LIN {X 0,Y 173.444,Z 1036.446,A -85,B 0,C 180,E1 -27586.228,E2 -27586.228} C_VEL
LIN {X 0,Y 162.464,Z 1044.017,A -85,B 0,C 180,E1 -27593.346,E2 -27593.346} C_VEL
LIN {X 0,Y 153.982,Z 1050.121,A -85,B 0,C 180,E1 -27601.28,E2 -27601.28} C_VEL
LIN {X 0,Y 148.005,Z 1054.743,A -85,B 0,C 180,E1 -27610.258,E2 -27610.258} C_VEL
LIN {X 0,Y 145.243,Z 1057.412,A -85,B 0,C 180,E1 -27618.081,E2 -27618.081} C_VEL
LIN {X 0,Y 144.199,Z 1058.976,A -85,B 0,C 180,E1 -27625.626,E2 -27625.626} C_VEL
LIN {X 0,Y 144.037,Z 1059.569,A -85,B 0,C 180,E1 -27632.387,E2 -27632.387} C_VEL
LIN {X 0,Y 144.314,Z 1059.398,A -85,B 0,C 180,E1 -27639.572,E2 -27639.572} C_VEL
LIN {X 0,Y 146.072,Z 1057.914,A -85,B 0,C 180,E1 -27648.767,E2 -27648.767} C_VEL
LIN {X 0,Y 149.888,Z 1055.271,A -85,B 0,C 180,E1 -27656.976,E2 -27656.976} C_VEL
LIN {X 0,Y 156.774,Z 1051.046,A -85,B 0,C 180,E1 -27665.478,E2 -27665.478} C_VEL
LIN {X 0,Y 166.876,Z 1044.865,A -85,B 0,C 180,E1 -27673.556,E2 -27673.556} C_VEL
LIN {X 0,Y 177.931,Z 1038.053,A -85,B 0,C 180,E1 -27679.841,E2 -27679.841} C_VEL
LIN {X 0,Y 192.704,Z 1028.454,A -85,B 0,C 180,E1 -27686.119,E2 -27686.119} C_VEL
LIN {X 0,Y 206.466,Z 1018.863,A -85,B 0,C 180,E1 -27690.659,E2 -27690.659} C_VEL
LIN {X 0,Y 223.283,Z 1006.192,A -85,B 0,C 180,E1 -27695.106,E2 -27695.106} C_VEL
LIN {X 0,Y 238.041,Z 993.951,A -85,B 0,C 180,E1 -27698.306,E2 -27698.306} C_VEL
LIN {X 0,Y 254.411,Z 979.174,A -85,B 0,C 180,E1 -27701.295,E2 -27701.295} C_VEL
LIN {X 0,Y 269.808,Z 963.547,A -85,B 0,C 180,E1 -27703.706,E2 -27703.706} C_VEL
LIN {X 0,Y 285.132,Z 946.472,A -85,B 0,C 180,E1 -27705.79,E2 -27705.79} C_VEL
LIN {X 0,Y 299.537,Z 928.245,A -85,B 0,C 180,E1 -27707.528,E2 -27707.528} C_VEL
LIN {X 0,Y 312.45,Z 910.056,A -85,B 0,C 180,E1 -27708.93,E2 -27708.93} C_VEL
LIN {X 0,Y 325.685,Z 888.747,A -85,B 0,C 180,E1 -27710.233,E2 -27710.233} C_VEL
LIN {X 0,Y 335.946,Z 869.895,A -85,B 0,C 180,E1 -27711.169,E2 -27711.169} C_VEL
LIN {X 0,Y 346.944,Z 846.425,A -85,B 0,C 180,E1 -27712.112,E2 -27712.112} C_VEL
LIN {X 0,Y 354.795,Z 826.568,A -85,B 0,C 180,E1 -27712.753,E2 -27712.753} C_VEL
LIN {X 0,Y 362.673,Z 802.827,A -85,B 0,C 180,E1 -27713.362,E2 -27713.362} C_VEL
LIN {X 0,Y 368.63,Z 779.656,A -85,B 0,C 180,E1 -27713.815,E2 -27713.815} C_VEL
LIN {X 0,Y 373.408,Z 755.336,A -85,B 0,C 180,E1 -27714.19,E2 -27714.19} C_VEL
LIN {X 0,Y 379.555,Z 704.729,A -85,B 0,C 180,E1 -27714.844,E2 -27714.844} C_VEL
LIN {X 0,Y 386.488,Z 644.435,A -85,B 0,C 180,E1 -27715.615,E2 -27715.615} C_VEL
LIN {X 0,Y 385.979,Z 642.999,A -85,B 0,C 180,E1 -27716.881,E2 -27716.881} C_VEL
LIN {X 0,Y 385.387,Z 640.321,A -85,B 0,C 180,E1 -27720.892,E2 -27720.892} C_VEL
LIN {X 0,Y 386.259,Z 643.666,A -85,B 0,C 180,E1 -27725.496,E2 -27725.496} C_VEL
LIN {X 0,Y 386.489,Z 644.784,A -85,B 0,C 180,E1 -27726.121,E2 -27726.121} C_VEL
LIN {X 0,Y 373.686,Z 754.037,A -85,B 0,C 180,E1 -27727.517,E2 -27727.517} C_VEL
LIN {X 0,Y 368.823,Z 780.194,A -85,B 0,C 180,E1 -27727.896,E2 -27727.896} C_VEL
LIN {X 0,Y 363.895,Z 799.826,A -85,B 0,C 180,E1 -27728.218,E2 -27728.218} C_VEL
LIN {X 0,Y 361.672,Z 807.261,A -85,B 0,C 180,E1 -27728.183,E2 -27728.183} C_VEL
LIN {X 0,Y 354.681,Z 825.951,A -85,B 0,C 180,E1 -27727.636,E2 -27727.636} C_VEL
LIN {X 0,Y 351.901,Z 833.043,A -85,B 0,C 180,E1 -27727.655,E2 -27727.655} C_VEL
LIN {X 0,Y 341.59,Z 857.457,A -85,B 0,C 180,E1 -27728.357,E2 -27728.357} C_VEL
LIN {X 0,Y 331.506,Z 877.698,A -85,B 0,C 180,E1 -27729.106,E2 -27729.106} C_VEL
LIN {X 0,Y 318.47,Z 900.334,A -85,B 0,C 180,E1 -27730.171,E2 -27730.171} C_VEL
LIN {X 0,Y 306.359,Z 918.658,A -85,B 0,C 180,E1 -27731.256,E2 -27731.256} C_VEL
LIN {X 0,Y 292.091,Z 937.956,A -85,B 0,C 180,E1 -27732.679,E2 -27732.679} C_VEL
LIN {X 0,Y 277.137,Z 955.733,A -85,B 0,C 180,E1 -27734.366,E2 -27734.366} C_VEL
LIN {X 0,Y 260.71,Z 973.388,A -85,B 0,C 180,E1 -27736.501,E2 -27736.501} C_VEL
LIN {X 0,Y 244.275,Z 989.022,A -85,B 0,C 180,E1 -27738.994,E2 -27738.994} C_VEL
LIN {X 0,Y 227.573,Z 1003.58,A -85,B 0,C 180,E1 -27742.017,E2 -27742.017} C_VEL
LIN {X 0,Y 210.824,Z 1016.635,A -85,B 0,C 180,E1 -27745.694,E2 -27745.694} C_VEL
LIN {X 0,Y 195.09,Z 1028.025,A -85,B 0,C 180,E1 -27749.983,E2 -27749.983} C_VEL
LIN {X 0,Y 179.302,Z 1038.497,A -85,B 0,C 180,E1 -27755.494,E2 -27755.494} C_VEL
LIN {X 0,Y 166.53,Z 1046.54,A -85,B 0,C 180,E1 -27761.363,E2 -27761.363} C_VEL
LIN {X 0,Y 153.385,Z 1054.528,A -85,B 0,C 180,E1 -27769.807,E2 -27769.807} C_VEL
LIN {X 0,Y 145.319,Z 1059.505,A -85,B 0,C 180,E1 -27777.541,E2 -27777.541} C_VEL
LIN {X 0,Y 139.028,Z 1063.816,A -85,B 0,C 180,E1 -27787.593,E2 -27787.593} C_VEL
LIN {X 0,Y 136.508,Z 1066.001,A -85,B 0,C 180,E1 -27796.444,E2 -27796.444} C_VEL
LIN {X 0,Y 135.999,Z 1066.928,A -85,B 0,C 180,E1 -27804.092,E2 -27804.092} C_VEL
LIN {X 0,Y 136.059,Z 1067.021,A -85,B 0,C 180,E1 -27810,E2 -27810} C_VEL
LIN {X 0,Y 136.006,Z 1066.417,A -85,B 0,C 180,E1 -27816.755,E2 -27816.755} C_VEL
LIN {X 0,Y 136.711,Z 1064.717,A -85,B 0,C 180,E1 -27824.832,E2 -27824.832} C_VEL
LIN {X 0,Y 139.354,Z 1061.814,A -85,B 0,C 180,E1 -27833.302,E2 -27833.302} C_VEL
LIN {X 0,Y 145.833,Z 1056.613,A -85,B 0,C 180,E1 -27843.265,E2 -27843.265} C_VEL
LIN {X 0,Y 154.501,Z 1050.4,A -85,B 0,C 180,E1 -27851.309,E2 -27851.309} C_VEL
LIN {X 0,Y 166.227,Z 1042.388,A -85,B 0,C 180,E1 -27858.755,E2 -27858.755} C_VEL
LIN {X 0,Y 179.96,Z 1032.608,A -85,B 0,C 180,E1 -27865.09,E2 -27865.09} C_VEL
LIN {X 0,Y 195.382,Z 1021.235,A -85,B 0,C 180,E1 -27870.458,E2 -27870.458} C_VEL
LIN {X 0,Y 211.129,Z 1008.531,A -85,B 0,C 180,E1 -27874.771,E2 -27874.771} C_VEL
LIN {X 0,Y 227.067,Z 994.761,A -85,B 0,C 180,E1 -27878.301,E2 -27878.301} C_VEL
LIN {X 0,Y 243.473,Z 978.966,A -85,B 0,C 180,E1 -27881.317,E2 -27881.317} C_VEL
LIN {X 0,Y 258.429,Z 963.247,A -85,B 0,C 180,E1 -27883.645,E2 -27883.645} C_VEL
LIN {X 0,Y 273.92,Z 944.994,A -85,B 0,C 180,E1 -27885.732,E2 -27885.732} C_VEL
LIN {X 0,Y 287.009,Z 927.872,A -85,B 0,C 180,E1 -27887.283,E2 -27887.283} C_VEL
LIN {X 0,Y 301.23,Z 906.903,A -85,B 0,C 180,E1 -27888.775,E2 -27888.775} C_VEL
LIN {X 0,Y 312.372,Z 888.252,A -85,B 0,C 180,E1 -27889.832,E2 -27889.832} C_VEL
LIN {X 0,Y 324.093,Z 865.864,A -85,B 0,C 180,E1 -27890.845,E2 -27890.845} C_VEL
LIN {X 0,Y 333.067,Z 845.762,A -85,B 0,C 180,E1 -27891.564,E2 -27891.564} C_VEL
LIN {X 0,Y 341.865,Z 822.855,A -85,B 0,C 180,E1 -27892.213,E2 -27892.213} C_VEL
LIN {X 0,Y 349.212,Z 798.837,A -85,B 0,C 180,E1 -27892.723,E2 -27892.723} C_VEL
LIN {X 0,Y 355.105,Z 774.615,A -85,B 0,C 180,E1 -27893.129,E2 -27893.129} C_VEL
LIN {X 0,Y 359.226,Z 749.857,A -85,B 0,C 180,E1 -27893.486,E2 -27893.486} C_VEL
LIN {X 0,Y 371.93,Z 639.67,A -85,B 0,C 180,E1 -27894.91,E2 -27894.91} C_VEL
LIN {X 0,Y 370.985,Z 636.993,A -85,B 0,C 180,E1 -27897.065,E2 -27897.065} C_VEL
LIN {X 0,Y 370.365,Z 634.188,A -85,B 0,C 180,E1 -27901.392,E2 -27901.392} C_VEL
LIN {X 0,Y 371.309,Z 637.843,A -85,B 0,C 180,E1 -27906.184,E2 -27906.184} C_VEL
LIN {X 0,Y 371.884,Z 639.748,A -85,B 0,C 180,E1 -27907.457,E2 -27907.457} C_VEL
LIN {X 0,Y 358.891,Z 751.554,A -85,B 0,C 180,E1 -27908.9,E2 -27908.9} C_VEL
LIN {X 0,Y 354.116,Z 777.471,A -85,B 0,C 180,E1 -27909.3,E2 -27909.3} C_VEL
LIN {X 0,Y 348.715,Z 799.063,A -85,B 0,C 180,E1 -27909.723,E2 -27909.723} C_VEL
LIN {X 0,Y 340.54,Z 824.701,A -85,B 0,C 180,E1 -27910.384,E2 -27910.384} C_VEL
LIN {X 0,Y 332.636,Z 845.015,A -85,B 0,C 180,E1 -27911.055,E2 -27911.055} C_VEL
LIN {X 0,Y 322.011,Z 868.172,A -85,B 0,C 180,E1 -27912.008,E2 -27912.008} C_VEL
LIN {X 0,Y 311.508,Z 887.711,A -85,B 0,C 180,E1 -27913.007,E2 -27913.007} C_VEL
LIN {X 0,Y 299.205,Z 907.957,A -85,B 0,C 180,E1 -27914.274,E2 -27914.274} C_VEL
LIN {X 0,Y 285.765,Z 927.152,A -85,B 0,C 180,E1 -27915.799,E2 -27915.799} C_VEL
LIN {X 0,Y 271.231,Z 945.815,A -85,B 0,C 180,E1 -27917.645,E2 -27917.645} C_VEL
LIN {X 0,Y 256.135,Z 962.851,A -85,B 0,C 180,E1 -27919.813,E2 -27919.813} C_VEL
LIN {X 0,Y 241.033,Z 978.385,A -85,B 0,C 180,E1 -27922.319,E2 -27922.319} C_VEL
LIN {X 0,Y 224.836,Z 993.303,A -85,B 0,C 180,E1 -27925.474,E2 -27925.474} C_VEL
LIN {X 0,Y 210.146,Z 1005.718,A -85,B 0,C 180,E1 -27928.898,E2 -27928.898} C_VEL
LIN {X 0,Y 193.459,Z 1018.601,A -85,B 0,C 180,E1 -27933.682,E2 -27933.682} C_VEL
LIN {X 0,Y 180.153,Z 1028.144,A -85,B 0,C 180,E1 -27938.502,E2 -27938.502} C_VEL
LIN {X 0,Y 165.451,Z 1038.099,A -85,B 0,C 180,E1 -27945.49,E2 -27945.49} C_VEL
LIN {X 0,Y 155.106,Z 1044.871,A -85,B 0,C 180,E1 -27952.236,E2 -27952.236} C_VEL
LIN {X 0,Y 145.923,Z 1051.053,A -85,B 0,C 180,E1 -27960.889,E2 -27960.889} C_VEL
LIN {X 0,Y 140.019,Z 1055.292,A -85,B 0,C 180,E1 -27969.954,E2 -27969.954} C_VEL
LIN {X 0,Y 137.097,Z 1057.973,A -85,B 0,C 180,E1 -27978.643,E2 -27978.643} C_VEL
LIN {X 0,Y 136.125,Z 1059.517,A -85,B 0,C 180,E1 -27987.474,E2 -27987.474} C_VEL
LIN {X 0,Y 136.078,Z 1059.854,A -85,B 0,C 180,E1 -27995.059,E2 -27995.059} C_VEL
LIN {X 0,Y 136.713,Z 1059.293,A -85,B 0,C 180,E1 -28003.105,E2 -28003.105} C_VEL
LIN {X 0,Y 138.991,Z 1057.679,A -85,B 0,C 180,E1 -28011.524,E2 -28011.524} C_VEL
LIN {X 0,Y 143.709,Z 1054.848,A -85,B 0,C 180,E1 -28020.063,E2 -28020.063} C_VEL
LIN {X 0,Y 152.977,Z 1049.573,A -85,B 0,C 180,E1 -28029.833,E2 -28029.833} C_VEL
LIN {X 0,Y 163.062,Z 1043.85,A -85,B 0,C 180,E1 -28036.862,E2 -28036.862} C_VEL
LIN {X 0,Y 177.76,Z 1035.167,A -85,B 0,C 180,E1 -28044.197,E2 -28044.197} C_VEL
LIN {X 0,Y 191.676,Z 1026.338,A -85,B 0,C 180,E1 -28049.399,E2 -28049.399} C_VEL
LIN {X 0,Y 208.569,Z 1014.772,A -85,B 0,C 180,E1 -28054.327,E2 -28054.327} C_VEL
LIN {X 0,Y 224.273,Z 1002.903,A -85,B 0,C 180,E1 -28058.006,E2 -28058.006} C_VEL
LIN {X 0,Y 240.811,Z 989.282,A -85,B 0,C 180,E1 -28061.208,E2 -28061.208} C_VEL
LIN {X 0,Y 256.218,Z 975.058,A -85,B 0,C 180,E1 -28063.743,E2 -28063.743} C_VEL
LIN {X 0,Y 271.177,Z 959.936,A -85,B 0,C 180,E1 -28065.869,E2 -28065.869} C_VEL
LIN {X 0,Y 286.867,Z 942.134,A -85,B 0,C 180,E1 -28067.826,E2 -28067.826} C_VEL
LIN {X 0,Y 299.674,Z 925.914,A -85,B 0,C 180,E1 -28069.253,E2 -28069.253} C_VEL
LIN {X 0,Y 314.092,Z 905.408,A -85,B 0,C 180,E1 -28070.702,E2 -28070.702} C_VEL
LIN {X 0,Y 325.346,Z 887.102,A -85,B 0,C 180,E1 -28071.732,E2 -28071.732} C_VEL
LIN {X 0,Y 336.695,Z 866.245,A -85,B 0,C 180,E1 -28072.697,E2 -28072.697} C_VEL
LIN {X 0,Y 346.692,Z 844.499,A -85,B 0,C 180,E1 -28073.498,E2 -28073.498} C_VEL
LIN {X 0,Y 354.828,Z 823.837,A -85,B 0,C 180,E1 -28074.12,E2 -28074.12} C_VEL
LIN {X 0,Y 362.88,Z 798.729,A -85,B 0,C 180,E1 -28074.711,E2 -28074.711} C_VEL
LIN {X 0,Y 368.398,Z 776.886,A -85,B 0,C 180,E1 -28075.103,E2 -28075.103} C_VEL
LIN {X 0,Y 373.276,Z 750.254,A -85,B 0,C 180,E1 -28075.481,E2 -28075.481} C_VEL
LIN {X 0,Y 385.06,Z 651.072,A -85,B 0,C 180,E1 -28076.725,E2 -28076.725} C_VEL
LIN {X 0,Y 384.406,Z 648.313,A -85,B 0,C 180,E1 -28080.894,E2 -28080.894} C_VEL
LIN {X 0,Y 385.072,Z 651.262,A -85,B 0,C 180,E1 -28085.014,E2 -28085.014} C_VEL
LIN {X 0,Y 372.858,Z 753.848,A -85,B 0,C 180,E1 -28086.29,E2 -28086.29} C_VEL
LIN {X 0,Y 367.945,Z 779.986,A -85,B 0,C 180,E1 -28086.654,E2 -28086.654} C_VEL
LIN {X 0,Y 362.317,Z 801.977,A -85,B 0,C 180,E1 -28087,E2 -28087} C_VEL
LIN {X 0,Y 354.003,Z 827.41,A -85,B 0,C 180,E1 -28087.516,E2 -28087.516} C_VEL
LIN {X 0,Y 351.901,Z 833.043,A -85,B 0,C 180,E1 -28087.655,E2 -28087.655} C_VEL
LIN {X 0,Y 348.96,Z 840.283,A -85,B 0,C 180,E1 -28087.682,E2 -28087.682} C_VEL
LIN {X 0,Y 340.298,Z 858.245,A -85,B 0,C 180,E1 -28087.209,E2 -28087.209} C_VEL
LIN {X 0,Y 336.89,Z 865.113,A -85,B 0,C 180,E1 -28087.266,E2 -28087.266} C_VEL
LIN {X 0,Y 325.209,Z 886.908,A -85,B 0,C 180,E1 -28088.1,E2 -28088.1} C_VEL
LIN {X 0,Y 313.827,Z 905.472,A -85,B 0,C 180,E1 -28088.997,E2 -28088.997} C_VEL
LIN {X 0,Y 299.256,Z 926.414,A -85,B 0,C 180,E1 -28090.264,E2 -28090.264} C_VEL
LIN {X 0,Y 285.785,Z 943.458,A -85,B 0,C 180,E1 -28091.579,E2 -28091.579} C_VEL
LIN {X 0,Y 270.221,Z 961.244,A -85,B 0,C 180,E1 -28093.303,E2 -28093.303} C_VEL
LIN {X 0,Y 254.044,Z 977.534,A -85,B 0,C 180,E1 -28095.357,E2 -28095.357} C_VEL
LIN {X 0,Y 238.257,Z 992.011,A -85,B 0,C 180,E1 -28097.703,E2 -28097.703} C_VEL
LIN {X 0,Y 220.432,Z 1006.67,A -85,B 0,C 180,E1 -28100.864,E2 -28100.864} C_VEL
LIN {X 0,Y 204.985,Z 1018.231,A -85,B 0,C 180,E1 -28104.194,E2 -28104.194} C_VEL
LIN {X 0,Y 186.511,Z 1030.839,A -85,B 0,C 180,E1 -28109.2,E2 -28109.2} C_VEL
LIN {X 0,Y 171.931,Z 1039.978,A -85,B 0,C 180,E1 -28114.328,E2 -28114.328} C_VEL
LIN {X 0,Y 156.524,Z 1049.055,A -85,B 0,C 180,E1 -28121.634,E2 -28121.634} C_VEL
LIN {X 0,Y 145.248,Z 1055.417,A -85,B 0,C 180,E1 -28129.222,E2 -28129.222} C_VEL
LIN {X 0,Y 135.786,Z 1060.915,A -85,B 0,C 180,E1 -28138.972,E2 -28138.972} C_VEL
LIN {X 0,Y 130.572,Z 1064.21,A -85,B 0,C 180,E1 -28148.434,E2 -28148.434} C_VEL
LIN {X 0,Y 128.359,Z 1066.085,A -85,B 0,C 180,E1 -28157.402,E2 -28157.402} C_VEL
LIN {X 0,Y 128.002,Z 1066.818,A -85,B 0,C 180,E1 -28165.52,E2 -28165.52} C_VEL
LIN {X 0,Y 128.037,Z 1066.713,A -85,B 0,C 180,E1 -28171.79,E2 -28171.79} C_VEL
LIN {X 0,Y 128.044,Z 1065.979,A -85,B 0,C 180,E1 -28178.532,E2 -28178.532} C_VEL
LIN {X 0,Y 129.155,Z 1064.128,A -85,B 0,C 180,E1 -28187.109,E2 -28187.109} C_VEL
LIN {X 0,Y 133.454,Z 1060.36,A -85,B 0,C 180,E1 -28197.68,E2 -28197.68} C_VEL
LIN {X 0,Y 140.894,Z 1055.047,A -85,B 0,C 180,E1 -28207.101,E2 -28207.101} C_VEL
LIN {X 0,Y 151.918,Z 1047.938,A -85,B 0,C 180,E1 -28215.841,E2 -28215.841} C_VEL
LIN {X 0,Y 165.139,Z 1039.209,A -85,B 0,C 180,E1 -28223.057,E2 -28223.057} C_VEL
LIN {X 0,Y 179.785,Z 1029.321,A -85,B 0,C 180,E1 -28228.924,E2 -28228.924} C_VEL
LIN {X 0,Y 195.964,Z 1017.429,A -85,B 0,C 180,E1 -28233.899,E2 -28233.899} C_VEL
LIN {X 0,Y 211.756,Z 1004.997,A -85,B 0,C 180,E1 -28237.743,E2 -28237.743} C_VEL
LIN {X 0,Y 228.856,Z 990.097,A -85,B 0,C 180,E1 -28241.137,E2 -28241.137} C_VEL
LIN {X 0,Y 243.866,Z 975.771,A -85,B 0,C 180,E1 -28243.625,E2 -28243.625} C_VEL
LIN {X 0,Y 260.896,Z 957.673,A -85,B 0,C 180,E1 -28246.028,E2 -28246.028} C_VEL
LIN {X 0,Y 274.295,Z 941.809,A -85,B 0,C 180,E1 -28247.672,E2 -28247.672} C_VEL
LIN {X 0,Y 289.489,Z 921.719,A -85,B 0,C 180,E1 -28249.313,E2 -28249.313} C_VEL
LIN {X 0,Y 302.091,Z 902.766,A -85,B 0,C 180,E1 -28250.522,E2 -28250.522} C_VEL
LIN {X 0,Y 314.82,Z 881.085,A -85,B 0,C 180,E1 -28251.628,E2 -28251.628} C_VEL
LIN {X 0,Y 325.282,Z 860.292,A -85,B 0,C 180,E1 -28252.454,E2 -28252.454} C_VEL
LIN {X 0,Y 334.797,Z 838.537,A -85,B 0,C 180,E1 -28253.139,E2 -28253.139} C_VEL
LIN {X 0,Y 343.033,Z 815.564,A -85,B 0,C 180,E1 -28253.701,E2 -28253.701} C_VEL
LIN {X 0,Y 349.627,Z 793.272,A -85,B 0,C 180,E1 -28254.123,E2 -28254.123} C_VEL
LIN {X 0,Y 355.299,Z 767.873,A -85,B 0,C 180,E1 -28254.509,E2 -28254.509} C_VEL
LIN {X 0,Y 358.865,Z 745.266,A -85,B 0,C 180,E1 -28254.818,E2 -28254.818} C_VEL
LIN {X 0,Y 370.36,Z 646.203,A -85,B 0,C 180,E1 -28256.091,E2 -28256.091} C_VEL
LIN {X 0,Y 369.892,Z 644.775,A -85,B 0,C 180,E1 -28257.366,E2 -28257.366} C_VEL
LIN {X 0,Y 369.384,Z 642.181,A -85,B 0,C 180,E1 -28261.396,E2 -28261.396} C_VEL
LIN {X 0,Y 370.228,Z 645.651,A -85,B 0,C 180,E1 -28265.968,E2 -28265.968} C_VEL
LIN {X 0,Y 370.338,Z 646.293,A -85,B 0,C 180,E1 -28266.307,E2 -28266.307} C_VEL
LIN {X 0,Y 357.88,Z 751.789,A -85,B 0,C 180,E1 -28267.631,E2 -28267.631} C_VEL
LIN {X 0,Y 353.035,Z 777.762,A -85,B 0,C 180,E1 -28268.015,E2 -28268.015} C_VEL
LIN {X 0,Y 347.557,Z 799.413,A -85,B 0,C 180,E1 -28268.42,E2 -28268.42} C_VEL
LIN {X 0,Y 339.664,Z 824.008,A -85,B 0,C 180,E1 -28269.021,E2 -28269.021} C_VEL
LIN {X 0,Y 331.666,Z 844.431,A -85,B 0,C 180,E1 -28269.66,E2 -28269.66} C_VEL
LIN {X 0,Y 321.374,Z 866.861,A -85,B 0,C 180,E1 -28270.527,E2 -28270.527} C_VEL
LIN {X 0,Y 310.217,Z 887.437,A -85,B 0,C 180,E1 -28271.521,E2 -28271.521} C_VEL
LIN {X 0,Y 297.782,Z 907.691,A -85,B 0,C 180,E1 -28272.725,E2 -28272.725} C_VEL
LIN {X 0,Y 284.128,Z 926.943,A -85,B 0,C 180,E1 -28274.181,E2 -28274.181} C_VEL
LIN {X 0,Y 269.735,Z 945.158,A -85,B 0,C 180,E1 -28275.896,E2 -28275.896} C_VEL
LIN {X 0,Y 254.375,Z 962.289,A -85,B 0,C 180,E1 -28277.965,E2 -28277.965} C_VEL
LIN {X 0,Y 239.451,Z 977.364,A -85,B 0,C 180,E1 -28280.279,E2 -28280.279} C_VEL
LIN {X 0,Y 222.273,Z 992.933,A -85,B 0,C 180,E1 -28283.41,E2 -28283.41} C_VEL
LIN {X 0,Y 207.108,Z 1005.405,A -85,B 0,C 180,E1 -28286.728,E2 -28286.728} C_VEL
LIN {X 0,Y 189.492,Z 1018.593,A -85,B 0,C 180,E1 -28291.493,E2 -28291.493} C_VEL
LIN {X 0,Y 175.853,Z 1027.98,A -85,B 0,C 180,E1 -28296.157,E2 -28296.157} C_VEL
LIN {X 0,Y 160.888,Z 1037.679,A -85,B 0,C 180,E1 -28302.832,E2 -28302.832} C_VEL
LIN {X 0,Y 149.223,Z 1044.838,A -85,B 0,C 180,E1 -28309.965,E2 -28309.965} C_VEL
LIN {X 0,Y 139.232,Z 1051.1,A -85,B 0,C 180,E1 -28318.864,E2 -28318.864} C_VEL
LIN {X 0,Y 132.661,Z 1055.377,A -85,B 0,C 180,E1 -28328.326,E2 -28328.326} C_VEL
LIN {X 0,Y 129.421,Z 1057.985,A -85,B 0,C 180,E1 -28337.053,E2 -28337.053} C_VEL
LIN {X 0,Y 128.164,Z 1059.622,A -85,B 0,C 180,E1 -28346.422,E2 -28346.422} C_VEL
LIN {X 0,Y 128.058,Z 1060.074,A -85,B 0,C 180,E1 -28354.03,E2 -28354.03} C_VEL
LIN {X 0,Y 128.626,Z 1059.693,A -85,B 0,C 180,E1 -28362.572,E2 -28362.572} C_VEL
LIN {X 0,Y 131.235,Z 1057.989,A -85,B 0,C 180,E1 -28372.393,E2 -28372.393} C_VEL
LIN {X 0,Y 136.337,Z 1055.198,A -85,B 0,C 180,E1 -28381.38,E2 -28381.38} C_VEL
LIN {X 0,Y 146.26,Z 1050.004,A -85,B 0,C 180,E1 -28391.539,E2 -28391.539} C_VEL
LIN {X 0,Y 157.505,Z 1044.026,A -85,B 0,C 180,E1 -28399.065,E2 -28399.065} C_VEL
LIN {X 0,Y 172.914,Z 1035.402,A -85,B 0,C 180,E1 -28406.376,E2 -28406.376} C_VEL
LIN {X 0,Y 187.59,Z 1026.49,A -85,B 0,C 180,E1 -28411.58,E2 -28411.58} C_VEL
LIN {X 0,Y 205.337,Z 1014.749,A -85,B 0,C 180,E1 -28416.465,E2 -28416.465} C_VEL
LIN {X 0,Y 221.332,Z 1003.013,A -85,B 0,C 180,E1 -28419.995,E2 -28419.995} C_VEL
LIN {X 0,Y 239.151,Z 988.614,A -85,B 0,C 180,E1 -28423.232,E2 -28423.232} C_VEL
LIN {X 0,Y 254.925,Z 974.31,A -85,B 0,C 180,E1 -28425.651,E2 -28425.651} C_VEL
LIN {X 0,Y 271.109,Z 958.165,A -85,B 0,C 180,E1 -28427.785,E2 -28427.785} C_VEL
LIN {X 0,Y 286.688,Z 940.467,A -85,B 0,C 180,E1 -28429.589,E2 -28429.589} C_VEL
LIN {X 0,Y 301.117,Z 922.247,A -85,B 0,C 180,E1 -28431.07,E2 -28431.07} C_VEL
LIN {X 0,Y 314.773,Z 902.473,A -85,B 0,C 180,E1 -28432.342,E2 -28432.342} C_VEL
LIN {X 0,Y 326.215,Z 883.786,A -85,B 0,C 180,E1 -28433.311,E2 -28433.311} C_VEL
LIN {X 0,Y 338.158,Z 861.218,A -85,B 0,C 180,E1 -28434.26,E2 -28434.26} C_VEL
LIN {X 0,Y 346.835,Z 842.123,A -85,B 0,C 180,E1 -28434.9,E2 -28434.9} C_VEL
LIN {X 0,Y 355.792,Z 819.009,A -85,B 0,C 180,E1 -28435.532,E2 -28435.532} C_VEL
LIN {X 0,Y 362.834,Z 796.266,A -85,B 0,C 180,E1 -28436.023,E2 -28436.023} C_VEL
LIN {X 0,Y 368.845,Z 771.9,A -85,B 0,C 180,E1 -28436.425,E2 -28436.425} C_VEL
LIN {X 0,Y 372.999,Z 747.535,A -85,B 0,C 180,E1 -28436.743,E2 -28436.743} C_VEL
LIN {X 0,Y 383.708,Z 658.313,A -85,B 0,C 180,E1 -28437.827,E2 -28437.827} C_VEL
LIN {X 0,Y 383.425,Z 656.303,A -85,B 0,C 180,E1 -28440.897,E2 -28440.897} C_VEL
LIN {X 0,Y 383.701,Z 658.574,A -85,B 0,C 180,E1 -28443.909,E2 -28443.909} C_VEL
LIN {X 0,Y 372.175,Z 753.847,A -85,B 0,C 180,E1 -28445.061,E2 -28445.061} C_VEL
LIN {X 0,Y 367.238,Z 779.789,A -85,B 0,C 180,E1 -28445.407,E2 -28445.407} C_VEL
LIN {X 0,Y 361.55,Z 801.82,A -85,B 0,C 180,E1 -28445.734,E2 -28445.734} C_VEL
LIN {X 0,Y 353.527,Z 826.276,A -85,B 0,C 180,E1 -28446.197,E2 -28446.197} C_VEL
LIN {X 0,Y 345.326,Z 846.818,A -85,B 0,C 180,E1 -28446.708,E2 -28446.708} C_VEL
LIN {X 0,Y 336.89,Z 865.113,A -85,B 0,C 180,E1 -28447.266,E2 -28447.266} C_VEL
LIN {X 0,Y 333.321,Z 872.023,A -85,B 0,C 180,E1 -28447.338,E2 -28447.338} C_VEL
LIN {X 0,Y 322.979,Z 889.144,A -85,B 0,C 180,E1 -28446.959,E2 -28446.959} C_VEL
LIN {X 0,Y 318.967,Z 895.72,A -85,B 0,C 180,E1 -28447.067,E2 -28447.067} C_VEL
LIN {X 0,Y 305.618,Z 915.782,A -85,B 0,C 180,E1 -28448.087,E2 -28448.087} C_VEL
LIN {X 0,Y 292.246,Z 933.68,A -85,B 0,C 180,E1 -28449.223,E2 -28449.223} C_VEL
LIN {X 0,Y 275.862,Z 953.045,A -85,B 0,C 180,E1 -28450.806,E2 -28450.806} C_VEL
LIN {X 0,Y 261.098,Z 968.605,A -85,B 0,C 180,E1 -28452.436,E2 -28452.436} C_VEL
LIN {X 0,Y 242.759,Z 985.909,A -85,B 0,C 180,E1 -28454.796,E2 -28454.796} C_VEL
LIN {X 0,Y 227.108,Z 999.111,A -85,B 0,C 180,E1 -28457.179,E2 -28457.179} C_VEL
LIN {X 0,Y 209.182,Z 1012.887,A -85,B 0,C 180,E1 -28460.466,E2 -28460.466} C_VEL
LIN {X 0,Y 192.07,Z 1024.608,A -85,B 0,C 180,E1 -28464.352,E2 -28464.352} C_VEL
LIN {X 0,Y 175.273,Z 1035.25,A -85,B 0,C 180,E1 -28469.211,E2 -28469.211} C_VEL
LIN {X 0,Y 159.287,Z 1044.401,A -85,B 0,C 180,E1 -28475.309,E2 -28475.309} C_VEL
LIN {X 0,Y 145.952,Z 1051.661,A -85,B 0,C 180,E1 -28482.278,E2 -28482.278} C_VEL
LIN {X 0,Y 133.714,Z 1058.058,A -85,B 0,C 180,E1 -28491.635,E2 -28491.635} C_VEL
LIN {X 0,Y 126.04,Z 1062.211,A -85,B 0,C 180,E1 -28501.058,E2 -28501.058} C_VEL
LIN {X 0,Y 121.175,Z 1065.293,A -85,B 0,C 180,E1 -28512.719,E2 -28512.719} C_VEL
LIN {X 0,Y 120.027,Z 1066.452,A -85,B 0,C 180,E1 -28522.34,E2 -28522.34} C_VEL
LIN {X 0,Y 120.054,Z 1066.61,A -85,B 0,C 180,E1 -28529.523,E2 -28529.523} C_VEL
LIN {X 0,Y 120.009,Z 1066.11,A -85,B 0,C 180,E1 -28536.698,E2 -28536.698} C_VEL
LIN {X 0,Y 120.942,Z 1064.37,A -85,B 0,C 180,E1 -28546.325,E2 -28546.325} C_VEL
LIN {X 0,Y 124.187,Z 1061.519,A -85,B 0,C 180,E1 -28555.771,E2 -28555.771} C_VEL
LIN {X 0,Y 131.549,Z 1056.624,A -85,B 0,C 180,E1 -28566.361,E2 -28566.361} C_VEL
LIN {X 0,Y 141.948,Z 1050.183,A -85,B 0,C 180,E1 -28575.353,E2 -28575.353} C_VEL
LIN {X 0,Y 155.148,Z 1042.232,A -85,B 0,C 180,E1 -28583.049,E2 -28583.049} C_VEL
LIN {X 0,Y 170.574,Z 1032.312,A -85,B 0,C 180,E1 -28589.508,E2 -28589.508} C_VEL
LIN {X 0,Y 187.057,Z 1021.134,A -85,B 0,C 180,E1 -28594.683,E2 -28594.683} C_VEL
LIN {X 0,Y 203.778,Z 1008.56,A -85,B 0,C 180,E1 -28598.793,E2 -28598.793} C_VEL
LIN {X 0,Y 219.791,Z 995.518,A -85,B 0,C 180,E1 -28601.98,E2 -28601.98} C_VEL
LIN {X 0,Y 237.218,Z 979.715,A -85,B 0,C 180,E1 -28604.851,E2 -28604.851} C_VEL
LIN {X 0,Y 252.175,Z 964.723,A -85,B 0,C 180,E1 -28606.938,E2 -28606.938} C_VEL
LIN {X 0,Y 269.422,Z 945.358,A -85,B 0,C 180,E1 -28609.003,E2 -28609.003} C_VEL
LIN {X 0,Y 282.917,Z 928.318,A -85,B 0,C 180,E1 -28610.417,E2 -28610.417} C_VEL
LIN {X 0,Y 298.008,Z 906.79,A -85,B 0,C 180,E1 -28611.809,E2 -28611.809} C_VEL
LIN {X 0,Y 309.442,Z 888.158,A -85,B 0,C 180,E1 -28612.76,E2 -28612.76} C_VEL
LIN {X 0,Y 320.947,Z 866.883,A -85,B 0,C 180,E1 -28613.629,E2 -28613.629} C_VEL
LIN {X 0,Y 330.595,Z 845.825,A -85,B 0,C 180,E1 -28614.306,E2 -28614.306} C_VEL
LIN {X 0,Y 339.323,Z 823.637,A -85,B 0,C 180,E1 -28614.868,E2 -28614.868} C_VEL
LIN {X 0,Y 346.988,Z 799.383,A -85,B 0,C 180,E1 -28615.331,E2 -28615.331} C_VEL
LIN {X 0,Y 352.715,Z 776.555,A -85,B 0,C 180,E1 -28615.676,E2 -28615.676} C_VEL
LIN {X 0,Y 357.229,Z 751.211,A -85,B 0,C 180,E1 -28616.017,E2 -28616.017} C_VEL
LIN {X 0,Y 368.955,Z 652.825,A -85,B 0,C 180,E1 -28617.243,E2 -28617.243} C_VEL
LIN {X 0,Y 368.401,Z 650.188,A -85,B 0,C 180,E1 -28621.4,E2 -28621.4} C_VEL
LIN {X 0,Y 368.922,Z 652.997,A -85,B 0,C 180,E1 -28625.149,E2 -28625.149} C_VEL
LIN {X 0,Y 357.03,Z 752.13,A -85,B 0,C 180,E1 -28626.356,E2 -28626.356} C_VEL
LIN {X 0,Y 352.162,Z 777.923,A -85,B 0,C 180,E1 -28626.721,E2 -28626.721} C_VEL
LIN {X 0,Y 346.624,Z 799.601,A -85,B 0,C 180,E1 -28627.106,E2 -28627.106} C_VEL
LIN {X 0,Y 338.504,Z 824.588,A -85,B 0,C 180,E1 -28627.687,E2 -28627.687} C_VEL
LIN {X 0,Y 330.419,Z 844.968,A -85,B 0,C 180,E1 -28628.294,E2 -28628.294} C_VEL
LIN {X 0,Y 320.007,Z 867.333,A -85,B 0,C 180,E1 -28629.117,E2 -28629.117} C_VEL
LIN {X 0,Y 309.183,Z 887.081,A -85,B 0,C 180,E1 -28630.021,E2 -28630.021} C_VEL
LIN {X 0,Y 296.578,Z 907.398,A -85,B 0,C 180,E1 -28631.163,E2 -28631.163} C_VEL
LIN {X 0,Y 282.72,Z 926.733,A -85,B 0,C 180,E1 -28632.546,E2 -28632.546} C_VEL
LIN {X 0,Y 268.801,Z 944.121,A -85,B 0,C 180,E1 -28634.094,E2 -28634.094} C_VEL
LIN {X 0,Y 252.885,Z 961.726,A -85,B 0,C 180,E1 -28636.095,E2 -28636.095} C_VEL
LIN {X 0,Y 237.947,Z 976.565,A -85,B 0,C 180,E1 -28638.252,E2 -28638.252} C_VEL
LIN {X 0,Y 219.788,Z 992.744,A -85,B 0,C 180,E1 -28641.343,E2 -28641.343} C_VEL
LIN {X 0,Y 204.377,Z 1005.091,A -85,B 0,C 180,E1 -28644.498,E2 -28644.498} C_VEL
LIN {X 0,Y 186.421,Z 1018.179,A -85,B 0,C 180,E1 -28649.042,E2 -28649.042} C_VEL
LIN {X 0,Y 171.165,Z 1028.266,A -85,B 0,C 180,E1 -28653.951,E2 -28653.951} C_VEL
LIN {X 0,Y 155.456,Z 1037.949,A -85,B 0,C 180,E1 -28660.626,E2 -28660.626} C_VEL
LIN {X 0,Y 143.079,Z 1045.101,A -85,B 0,C 180,E1 -28667.865,E2 -28667.865} C_VEL
LIN {X 0,Y 132.341,Z 1051.348,A -85,B 0,C 180,E1 -28677.045,E2 -28677.045} C_VEL
LIN {X 0,Y 125.175,Z 1055.616,A -85,B 0,C 180,E1 -28686.958,E2 -28686.958} C_VEL
LIN {X 0,Y 121.589,Z 1058.217,A -85,B 0,C 180,E1 -28696.203,E2 -28696.203} C_VEL
LIN {X 0,Y 120.176,Z 1059.846,A -85,B 0,C 180,E1 -28706.184,E2 -28706.184} C_VEL
LIN {X 0,Y 120.057,Z 1060.267,A -85,B 0,C 180,E1 -28713.82,E2 -28713.82} C_VEL
LIN {X 0,Y 120.6,Z 1059.997,A -85,B 0,C 180,E1 -28722.449,E2 -28722.449} C_VEL
LIN {X 0,Y 123.513,Z 1058.299,A -85,B 0,C 180,E1 -28733.371,E2 -28733.371} C_VEL
LIN {X 0,Y 129.043,Z 1055.548,A -85,B 0,C 180,E1 -28742.847,E2 -28742.847} C_VEL
LIN {X 0,Y 139.206,Z 1050.684,A -85,B 0,C 180,E1 -28753.029,E2 -28753.029} C_VEL
LIN {X 0,Y 151.012,Z 1044.796,A -85,B 0,C 180,E1 -28760.777,E2 -28760.777} C_VEL
LIN {X 0,Y 166.39,Z 1036.761,A -85,B 0,C 180,E1 -28767.921,E2 -28767.921} C_VEL
LIN {X 0,Y 182.271,Z 1027.55,A -85,B 0,C 180,E1 -28773.403,E2 -28773.403} C_VEL
LIN {X 0,Y 199.512,Z 1016.739,A -85,B 0,C 180,E1 -28777.996,E2 -28777.996} C_VEL
LIN {X 0,Y 217.197,Z 1004.209,A -85,B 0,C 180,E1 -28781.757,E2 -28781.757} C_VEL
LIN {X 0,Y 235.133,Z 990.253,A -85,B 0,C 180,E1 -28784.863,E2 -28784.863} C_VEL
LIN {X 0,Y 252.107,Z 975.246,A -85,B 0,C 180,E1 -28787.335,E2 -28787.335} C_VEL
LIN {X 0,Y 267.644,Z 960.101,A -85,B 0,C 180,E1 -28789.277,E2 -28789.277} C_VEL
LIN {X 0,Y 283.449,Z 942.74,A -85,B 0,C 180,E1 -28791.013,E2 -28791.013} C_VEL
LIN {X 0,Y 296.637,Z 926.541,A -85,B 0,C 180,E1 -28792.307,E2 -28792.307} C_VEL
LIN {X 0,Y 311.398,Z 906.15,A -85,B 0,C 180,E1 -28793.614,E2 -28793.614} C_VEL
LIN {X 0,Y 323.41,Z 887.065,A -85,B 0,C 180,E1 -28794.581,E2 -28794.581} C_VEL
LIN {X 0,Y 335.02,Z 866.15,A -85,B 0,C 180,E1 -28795.448,E2 -28795.448} C_VEL
LIN {X 0,Y 345.477,Z 843.714,A -85,B 0,C 180,E1 -28796.183,E2 -28796.183} C_VEL
LIN {X 0,Y 354.205,Z 821.776,A -85,B 0,C 180,E1 -28796.763,E2 -28796.763} C_VEL
LIN {X 0,Y 361.842,Z 797.83,A -85,B 0,C 180,E1 -28797.261,E2 -28797.261} C_VEL
LIN {X 0,Y 367.588,Z 775.195,A -85,B 0,C 180,E1 -28797.623,E2 -28797.623} C_VEL
LIN {X 0,Y 372.198,Z 749.776,A -85,B 0,C 180,E1 -28797.946,E2 -28797.946} C_VEL
LIN {X 0,Y 382.496,Z 665.556,A -85,B 0,C 180,E1 -28798.951,E2 -28798.951} C_VEL
LIN {X 0,Y 382.444,Z 664.293,A -85,B 0,C 180,E1 -28800.899,E2 -28800.899} C_VEL
LIN {X 0,Y 382.492,Z 665.732,A -85,B 0,C 180,E1 -28802.795,E2 -28802.795} C_VEL
LIN {X 0,Y 371.661,Z 753.865,A -85,B 0,C 180,E1 -28803.829,E2 -28803.829} C_VEL
LIN {X 0,Y 366.66,Z 779.786,A -85,B 0,C 180,E1 -28804.158,E2 -28804.158} C_VEL
LIN {X 0,Y 360.9,Z 801.879,A -85,B 0,C 180,E1 -28804.466,E2 -28804.466} C_VEL
LIN {X 0,Y 352.752,Z 826.425,A -85,B 0,C 180,E1 -28804.902,E2 -28804.902} C_VEL
LIN {X 0,Y 344.162,Z 847.662,A -85,B 0,C 180,E1 -28805.4,E2 -28805.4} C_VEL
LIN {X 0,Y 332.852,Z 871.234,A -85,B 0,C 180,E1 -28806.106,E2 -28806.106} C_VEL
LIN {X 0,Y 322.247,Z 890.168,A -85,B 0,C 180,E1 -28806.823,E2 -28806.823} C_VEL
LIN {X 0,Y 318.967,Z 895.72,A -85,B 0,C 180,E1 -28807.067,E2 -28807.067} C_VEL
LIN {X 0,Y 314.839,Z 902.269,A -85,B 0,C 180,E1 -28807.189,E2 -28807.189} C_VEL
LIN {X 0,Y 302.975,Z 918.46,A -85,B 0,C 180,E1 -28806.906,E2 -28806.906} C_VEL
LIN {X 0,Y 298.214,Z 924.524,A -85,B 0,C 180,E1 -28807.068,E2 -28807.068} C_VEL
LIN {X 0,Y 283.914,Z 942.227,A -85,B 0,C 180,E1 -28808.26,E2 -28808.26} C_VEL
LIN {X 0,Y 268.808,Z 959.07,A -85,B 0,C 180,E1 -28809.692,E2 -28809.692} C_VEL
LIN {X 0,Y 251.122,Z 976.489,A -85,B 0,C 180,E1 -28811.622,E2 -28811.622} C_VEL
LIN {X 0,Y 235.585,Z 990.243,A -85,B 0,C 180,E1 -28813.605,E2 -28813.605} C_VEL
LIN {X 0,Y 215.985,Z 1005.771,A -85,B 0,C 180,E1 -28816.605,E2 -28816.605} C_VEL
LIN {X 0,Y 199.626,Z 1017.375,A -85,B 0,C 180,E1 -28819.668,E2 -28819.668} C_VEL
LIN {X 0,Y 180.741,Z 1029.519,A -85,B 0,C 180,E1 -28824.103,E2 -28824.103} C_VEL
LIN {X 0,Y 164.156,Z 1039.091,A -85,B 0,C 180,E1 -28829.163,E2 -28829.163} C_VEL
LIN {X 0,Y 147.965,Z 1047.771,A -85,B 0,C 180,E1 -28835.815,E2 -28835.815} C_VEL
LIN {X 0,Y 134.062,Z 1054.604,A -85,B 0,C 180,E1 -28843.919,E2 -28843.919} C_VEL
LIN {X 0,Y 122.722,Z 1060.188,A -85,B 0,C 180,E1 -28854.082,E2 -28854.082} C_VEL
LIN {X 0,Y 115.501,Z 1063.804,A -85,B 0,C 180,E1 -28865.447,E2 -28865.447} C_VEL
LIN {X 0,Y 112.579,Z 1065.671,A -85,B 0,C 180,E1 -28875.6,E2 -28875.6} C_VEL
LIN {X 0,Y 112.006,Z 1066.421,A -85,B 0,C 180,E1 -28885.392,E2 -28885.392} C_VEL
LIN {X 0,Y 112.038,Z 1066.28,A -85,B 0,C 180,E1 -28892.046,E2 -28892.046} C_VEL
LIN {X 0,Y 112.075,Z 1065.601,A -85,B 0,C 180,E1 -28899.241,E2 -28899.241} C_VEL
LIN {X 0,Y 113.391,Z 1063.899,A -85,B 0,C 180,E1 -28908.509,E2 -28908.509} C_VEL
LIN {X 0,Y 117.932,Z 1060.613,A -85,B 0,C 180,E1 -28919.456,E2 -28919.456} C_VEL
LIN {X 0,Y 126.723,Z 1055.319,A -85,B 0,C 180,E1 -28930.317,E2 -28930.317} C_VEL
LIN {X 0,Y 137.945,Z 1048.984,A -85,B 0,C 180,E1 -28938.924,E2 -28938.924} C_VEL
LIN {X 0,Y 153.657,Z 1039.893,A -85,B 0,C 180,E1 -28947.081,E2 -28947.081} C_VEL
LIN {X 0,Y 168.008,Z 1031.088,A -85,B 0,C 180,E1 -28952.469,E2 -28952.469} C_VEL
LIN {X 0,Y 185.99,Z 1019.157,A -85,B 0,C 180,E1 -28957.62,E2 -28957.62} C_VEL
LIN {X 0,Y 202.629,Z 1006.956,A -85,B 0,C 180,E1 -28961.341,E2 -28961.341} C_VEL
LIN {X 0,Y 220.875,Z 992.242,A -85,B 0,C 180,E1 -28964.631,E2 -28964.631} C_VEL
LIN {X 0,Y 237.01,Z 977.66,A -85,B 0,C 180,E1 -28967.041,E2 -28967.041} C_VEL
LIN {X 0,Y 253.983,Z 960.747,A -85,B 0,C 180,E1 -28969.186,E2 -28969.186} C_VEL
LIN {X 0,Y 269.384,Z 943.299,A -85,B 0,C 180,E1 -28970.869,E2 -28970.869} C_VEL
LIN {X 0,Y 284.049,Z 924.85,A -85,B 0,C 180,E1 -28972.271,E2 -28972.271} C_VEL
LIN {X 0,Y 297.961,Z 904.806,A -85,B 0,C 180,E1 -28973.448,E2 -28973.448} C_VEL
LIN {X 0,Y 309.928,Z 885.325,A -85,B 0,C 180,E1 -28974.365,E2 -28974.365} C_VEL
LIN {X 0,Y 322.091,Z 862.325,A -85,B 0,C 180,E1 -28975.207,E2 -28975.207} C_VEL
LIN {X 0,Y 330.868,Z 843.009,A -85,B 0,C 180,E1 -28975.762,E2 -28975.762} C_VEL
LIN {X 0,Y 340.118,Z 818.907,A -85,B 0,C 180,E1 -28976.31,E2 -28976.31} C_VEL
LIN {X 0,Y 346.949,Z 796.809,A -85,B 0,C 180,E1 -28976.69,E2 -28976.69} C_VEL
LIN {X 0,Y 352.996,Z 771.961,A -85,B 0,C 180,E1 -28977.036,E2 -28977.036} C_VEL
LIN {X 0,Y 356.987,Z 748.391,A -85,B 0,C 180,E1 -28977.334,E2 -28977.334} C_VEL
LIN {X 0,Y 367.625,Z 660.061,A -85,B 0,C 180,E1 -28978.402,E2 -28978.402} C_VEL
LIN {X 0,Y 367.418,Z 658.194,A -85,B 0,C 180,E1 -28981.403,E2 -28981.403} C_VEL
LIN {X 0,Y 367.593,Z 660.258,A -85,B 0,C 180,E1 -28983.989,E2 -28983.989} C_VEL
LIN {X 0,Y 356.344,Z 752.576,A -85,B 0,C 180,E1 -28985.078,E2 -28985.078} C_VEL
LIN {X 0,Y 351.41,Z 778.343,A -85,B 0,C 180,E1 -28985.425,E2 -28985.425} C_VEL
LIN {X 0,Y 345.789,Z 800.094,A -85,B 0,C 180,E1 -28985.791,E2 -28985.791} C_VEL
LIN {X 0,Y 337.529,Z 825.168,A -85,B 0,C 180,E1 -28986.344,E2 -28986.344} C_VEL
LIN {X 0,Y 329.361,Z 845.504,A -85,B 0,C 180,E1 -28986.918,E2 -28986.918} C_VEL
LIN {X 0,Y 318.359,Z 868.696,A -85,B 0,C 180,E1 -28987.731,E2 -28987.731} C_VEL
LIN {X 0,Y 307.414,Z 888.331,A -85,B 0,C 180,E1 -28988.59,E2 -28988.59} C_VEL
LIN {X 0,Y 294.186,Z 909.18,A -85,B 0,C 180,E1 -28989.715,E2 -28989.715} C_VEL
LIN {X 0,Y 280.149,Z 928.327,A -85,B 0,C 180,E1 -28991.035,E2 -28991.035} C_VEL
LIN {X 0,Y 264.823,Z 946.994,A -85,B 0,C 180,E1 -28992.65,E2 -28992.65} C_VEL
LIN {X 0,Y 248.953,Z 963.905,A -85,B 0,C 180,E1 -28994.546,E2 -28994.546} C_VEL
LIN {X 0,Y 231.999,Z 980.229,A -85,B 0,C 180,E1 -28996.904,E2 -28996.904} C_VEL
LIN {X 0,Y 214.615,Z 994.953,A -85,B 0,C 180,E1 -28999.76,E2 -28999.76} C_VEL
LIN {X 0,Y 197.025,Z 1008.519,A -85,B 0,C 180,E1 -29003.283,E2 -29003.283} C_VEL
LIN {X 0,Y 179.49,Z 1020.493,A -85,B 0,C 180,E1 -29007.657,E2 -29007.657} C_VEL
LIN {X 0,Y 163.159,Z 1030.799,A -85,B 0,C 180,E1 -29012.905,E2 -29012.905} C_VEL
LIN {X 0,Y 147.671,Z 1039.631,A -85,B 0,C 180,E1 -29019.53,E2 -29019.53} C_VEL
LIN {X 0,Y 135.006,Z 1046.546,A -85,B 0,C 180,E1 -29027.049,E2 -29027.049} C_VEL
LIN {X 0,Y 123.605,Z 1052.596,A -85,B 0,C 180,E1 -29037.181,E2 -29037.181} C_VEL
LIN {X 0,Y 117.004,Z 1056.319,A -85,B 0,C 180,E1 -29046.852,E2 -29046.852} C_VEL
LIN {X 0,Y 113.087,Z 1059.089,A -85,B 0,C 180,E1 -29058.267,E2 -29058.267} C_VEL
LIN {X 0,Y 112.1,Z 1060.233,A -85,B 0,C 180,E1 -29068.467,E2 -29068.467} C_VEL
LIN {X 0,Y 112.139,Z 1060.466,A -85,B 0,C 180,E1 -29076.656,E2 -29076.656} C_VEL
LIN {X 0,Y 113.251,Z 1059.849,A -85,B 0,C 180,E1 -29086.411,E2 -29086.411} C_VEL
LIN {X 0,Y 116.739,Z 1058.174,A -85,B 0,C 180,E1 -29096.448,E2 -29096.448} C_VEL
LIN {X 0,Y 124.512,Z 1054.812,A -85,B 0,C 180,E1 -29107.612,E2 -29107.612} C_VEL
LIN {X 0,Y 135.935,Z 1049.623,A -85,B 0,C 180,E1 -29117.355,E2 -29117.355} C_VEL
LIN {X 0,Y 150.415,Z 1042.886,A -85,B 0,C 180,E1 -29125.517,E2 -29125.517} C_VEL
LIN {X 0,Y 166.507,Z 1034.524,A -85,B 0,C 180,E1 -29131.976,E2 -29131.976} C_VEL
LIN {X 0,Y 183.473,Z 1024.981,A -85,B 0,C 180,E1 -29137.075,E2 -29137.075} C_VEL
LIN {X 0,Y 201.597,Z 1013.472,A -85,B 0,C 180,E1 -29141.322,E2 -29141.322} C_VEL
LIN {X 0,Y 217.988,Z 1002.004,A -85,B 0,C 180,E1 -29144.419,E2 -29144.419} C_VEL
LIN {X 0,Y 236.723,Z 987.299,A -85,B 0,C 180,E1 -29147.348,E2 -29147.348} C_VEL
LIN {X 0,Y 252.276,Z 973.658,A -85,B 0,C 180,E1 -29149.402,E2 -29149.402} C_VEL
LIN {X 0,Y 269.993,Z 956.293,A -85,B 0,C 180,E1 -29151.419,E2 -29151.419} C_VEL
LIN {X 0,Y 284.664,Z 940.026,A -85,B 0,C 180,E1 -29152.88,E2 -29152.88} C_VEL
LIN {X 0,Y 299.5,Z 921.709,A -85,B 0,C 180,E1 -29154.2,E2 -29154.2} C_VEL
LIN {X 0,Y 313.488,Z 901.774,A -85,B 0,C 180,E1 -29155.328,E2 -29155.328} C_VEL
LIN {X 0,Y 326.161,Z 881.362,A -85,B 0,C 180,E1 -29156.255,E2 -29156.255} C_VEL
LIN {X 0,Y 337.414,Z 860.061,A -85,B 0,C 180,E1 -29157.036,E2 -29157.036} C_VEL
LIN {X 0,Y 346.758,Z 839.635,A -85,B 0,C 180,E1 -29157.633,E2 -29157.633} C_VEL
LIN {X 0,Y 355.888,Z 815.615,A -85,B 0,C 180,E1 -29158.192,E2 -29158.192} C_VEL
LIN {X 0,Y 362.296,Z 794.911,A -85,B 0,C 180,E1 -29158.58,E2 -29158.58} C_VEL
LIN {X 0,Y 368.454,Z 769.446,A -85,B 0,C 180,E1 -29158.948,E2 -29158.948} C_VEL
LIN {X 0,Y 372.322,Z 746.73,A -85,B 0,C 180,E1 -29159.215,E2 -29159.215} C_VEL
LIN {X 0,Y 381.439,Z 672.756,A -85,B 0,C 180,E1 -29160.068,E2 -29160.068} C_VEL
LIN {X 0,Y 381.452,Z 672.386,A -85,B 0,C 180,E1 -29161.051,E2 -29161.051} C_VEL
LIN {X 0,Y 381.42,Z 672.966,A -85,B 0,C 180,E1 -29161.675,E2 -29161.675} C_VEL
LIN {X 0,Y 371.322,Z 753.862,A -85,B 0,C 180,E1 -29162.593,E2 -29162.593} C_VEL
LIN {X 0,Y 366.297,Z 779.61,A -85,B 0,C 180,E1 -29162.903,E2 -29162.903} C_VEL
LIN {X 0,Y 360.488,Z 801.723,A -85,B 0,C 180,E1 -29163.192,E2 -29163.192} C_VEL
LIN {X 0,Y 352.157,Z 826.574,A -85,B 0,C 180,E1 -29163.602,E2 -29163.602} C_VEL
LIN {X 0,Y 343.82,Z 847.028,A -85,B 0,C 180,E1 -29164.049,E2 -29164.049} C_VEL
LIN {X 0,Y 332.579,Z 870.374,A -85,B 0,C 180,E1 -29164.695,E2 -29164.695} C_VEL
LIN {X 0,Y 321.873,Z 889.371,A -85,B 0,C 180,E1 -29165.361,E2 -29165.361} C_VEL
LIN {X 0,Y 308.812,Z 909.865,A -85,B 0,C 180,E1 -29166.267,E2 -29166.267} C_VEL
LIN {X 0,Y 298.214,Z 924.524,A -85,B 0,C 180,E1 -29167.068,E2 -29167.068} C_VEL
LIN {X 0,Y 293.35,Z 930.543,A -85,B 0,C 180,E1 -29167.247,E2 -29167.247} C_VEL
LIN {X 0,Y 280.073,Z 945.634,A -85,B 0,C 180,E1 -29167.076,E2 -29167.076} C_VEL
LIN {X 0,Y 274.85,Z 951.224,A -85,B 0,C 180,E1 -29167.306,E2 -29167.306} C_VEL
LIN {X 0,Y 259.962,Z 966.576,A -85,B 0,C 180,E1 -29168.699,E2 -29168.699} C_VEL
LIN {X 0,Y 243.062,Z 982.334,A -85,B 0,C 180,E1 -29170.523,E2 -29170.523} C_VEL
LIN {X 0,Y 224.624,Z 997.462,A -85,B 0,C 180,E1 -29172.875,E2 -29172.875} C_VEL
LIN {X 0,Y 207.534,Z 1010.121,A -85,B 0,C 180,E1 -29175.509,E2 -29175.509} C_VEL
LIN {X 0,Y 187.816,Z 1023.112,A -85,B 0,C 180,E1 -29179.273,E2 -29179.273} C_VEL
LIN {X 0,Y 171.005,Z 1033.081,A -85,B 0,C 180,E1 -29183.364,E2 -29183.364} C_VEL
LIN {X 0,Y 151.605,Z 1043.422,A -85,B 0,C 180,E1 -29189.647,E2 -29189.647} C_VEL
LIN {X 0,Y 136.803,Z 1050.604,A -85,B 0,C 180,E1 -29196.301,E2 -29196.301} C_VEL
LIN {X 0,Y 121.687,Z 1057.462,A -85,B 0,C 180,E1 -29206.352,E2 -29206.352} C_VEL
LIN {X 0,Y 112.63,Z 1061.485,A -85,B 0,C 180,E1 -29215.993,E2 -29215.993} C_VEL
LIN {X 0,Y 106.212,Z 1064.656,A -85,B 0,C 180,E1 -29228.46,E2 -29228.46} C_VEL
LIN {X 0,Y 104.081,Z 1066.001,A -85,B 0,C 180,E1 -29240.601,E2 -29240.601} C_VEL
LIN {X 0,Y 104.052,Z 1066.199,A -85,B 0,C 180,E1 -29248.899,E2 -29248.899} C_VEL
LIN {X 0,Y 104.011,Z 1065.803,A -85,B 0,C 180,E1 -29256.624,E2 -29256.624} C_VEL
LIN {X 0,Y 105.268,Z 1064.022,A -85,B 0,C 180,E1 -29268.267,E2 -29268.267} C_VEL
LIN {X 0,Y 109.344,Z 1061.202,A -85,B 0,C 180,E1 -29278.99,E2 -29278.99} C_VEL
LIN {X 0,Y 118.19,Z 1056.373,A -85,B 0,C 180,E1 -29290.649,E2 -29290.649} C_VEL
LIN {X 0,Y 130.239,Z 1049.966,A -85,B 0,C 180,E1 -29300.151,E2 -29300.151} C_VEL
LIN {X 0,Y 145.069,Z 1042.054,A -85,B 0,C 180,E1 -29307.971,E2 -29307.971} C_VEL
LIN {X 0,Y 162,Z 1032.205,A -85,B 0,C 180,E1 -29314.308,E2 -29314.308} C_VEL
LIN {X 0,Y 178.876,Z 1021.623,A -85,B 0,C 180,E1 -29319.038,E2 -29319.038} C_VEL
LIN {X 0,Y 197.515,Z 1008.582,A -85,B 0,C 180,E1 -29323.094,E2 -29323.094} C_VEL
LIN {X 0,Y 214.32,Z 995.612,A -85,B 0,C 180,E1 -29326.025,E2 -29326.025} C_VEL
LIN {X 0,Y 232.528,Z 979.889,A -85,B 0,C 180,E1 -29328.642,E2 -29328.642} C_VEL
LIN {X 0,Y 247.507,Z 965.482,A -85,B 0,C 180,E1 -29330.466,E2 -29330.466} C_VEL
LIN {X 0,Y 264.395,Z 947.414,A -85,B 0,C 180,E1 -29332.235,E2 -29332.235} C_VEL
LIN {X 0,Y 279.214,Z 929.377,A -85,B 0,C 180,E1 -29333.592,E2 -29333.592} C_VEL
LIN {X 0,Y 293.651,Z 909.717,A -85,B 0,C 180,E1 -29334.746,E2 -29334.746} C_VEL
LIN {X 0,Y 306.829,Z 888.911,A -85,B 0,C 180,E1 -29335.702,E2 -29335.702} C_VEL
LIN {X 0,Y 318.904,Z 867.214,A -85,B 0,C 180,E1 -29336.483,E2 -29336.483} C_VEL
LIN {X 0,Y 328.89,Z 845.887,A -85,B 0,C 180,E1 -29337.081,E2 -29337.081} C_VEL
LIN {X 0,Y 337.766,Z 823.768,A -85,B 0,C 180,E1 -29337.57,E2 -29337.57} C_VEL
LIN {X 0,Y 345.646,Z 799.384,A -85,B 0,C 180,E1 -29337.975,E2 -29337.975} C_VEL
LIN {X 0,Y 351.371,Z 777.037,A -85,B 0,C 180,E1 -29338.271,E2 -29338.271} C_VEL
LIN {X 0,Y 356.147,Z 751.089,A -85,B 0,C 180,E1 -29338.588,E2 -29338.588} C_VEL
LIN {X 0,Y 366.455,Z 667.232,A -85,B 0,C 180,E1 -29339.57,E2 -29339.57} C_VEL
LIN {X 0,Y 366.435,Z 666.197,A -85,B 0,C 180,E1 -29341.407,E2 -29341.407} C_VEL
LIN {X 0,Y 366.428,Z 667.409,A -85,B 0,C 180,E1 -29342.82,E2 -29342.82} C_VEL
LIN {X 0,Y 355.85,Z 752.917,A -85,B 0,C 180,E1 -29343.794,E2 -29343.794} C_VEL
LIN {X 0,Y 350.903,Z 778.492,A -85,B 0,C 180,E1 -29344.121,E2 -29344.121} C_VEL
LIN {X 0,Y 345.228,Z 800.264,A -85,B 0,C 180,E1 -29344.465,E2 -29344.465} C_VEL
LIN {X 0,Y 336.741,Z 825.748,A -85,B 0,C 180,E1 -29344.994,E2 -29344.994} C_VEL
LIN {X 0,Y 328.495,Z 846.041,A -85,B 0,C 180,E1 -29345.534,E2 -29345.534} C_VEL
LIN {X 0,Y 317.38,Z 869.168,A -85,B 0,C 180,E1 -29346.298,E2 -29346.298} C_VEL
LIN {X 0,Y 306.319,Z 888.777,A -85,B 0,C 180,E1 -29347.105,E2 -29347.105} C_VEL
LIN {X 0,Y 292.936,Z 909.586,A -85,B 0,C 180,E1 -29348.164,E2 -29348.164} C_VEL
LIN {X 0,Y 279.066,Z 928.274,A -85,B 0,C 180,E1 -29349.377,E2 -29349.377} C_VEL
LIN {X 0,Y 263.71,Z 946.77,A -85,B 0,C 180,E1 -29350.879,E2 -29350.879} C_VEL
LIN {X 0,Y 247.964,Z 963.341,A -85,B 0,C 180,E1 -29352.621,E2 -29352.621} C_VEL
LIN {X 0,Y 232.474,Z 978.078,A -85,B 0,C 180,E1 -29354.593,E2 -29354.593} C_VEL
LIN {X 0,Y 213.759,Z 993.892,A -85,B 0,C 180,E1 -29357.4,E2 -29357.4} C_VEL
LIN {X 0,Y 197.329,Z 1006.337,A -85,B 0,C 180,E1 -29360.378,E2 -29360.378} C_VEL
LIN {X 0,Y 178.265,Z 1019.27,A -85,B 0,C 180,E1 -29364.679,E2 -29364.679} C_VEL
LIN {X 0,Y 162.616,Z 1028.836,A -85,B 0,C 180,E1 -29369.176,E2 -29369.176} C_VEL
LIN {X 0,Y 145.087,Z 1038.627,A -85,B 0,C 180,E1 -29375.859,E2 -29375.859} C_VEL
LIN {X 0,Y 131.446,Z 1045.626,A -85,B 0,C 180,E1 -29383.092,E2 -29383.092} C_VEL
LIN {X 0,Y 119.026,Z 1051.843,A -85,B 0,C 180,E1 -29392.783,E2 -29392.783} C_VEL
LIN {X 0,Y 110.456,Z 1056.096,A -85,B 0,C 180,E1 -29403.668,E2 -29403.668} C_VEL
LIN {X 0,Y 106.007,Z 1058.689,A -85,B 0,C 180,E1 -29414.176,E2 -29414.176} C_VEL
LIN {X 0,Y 104.206,Z 1060.293,A -85,B 0,C 180,E1 -29425.598,E2 -29425.598} C_VEL
LIN {X 0,Y 104.07,Z 1060.702,A -85,B 0,C 180,E1 -29434.408,E2 -29434.408} C_VEL
LIN {X 0,Y 104.839,Z 1060.422,A -85,B 0,C 180,E1 -29444.358,E2 -29444.358} C_VEL
LIN {X 0,Y 108.699,Z 1058.693,A -85,B 0,C 180,E1 -29456.839,E2 -29456.839} C_VEL
LIN {X 0,Y 115.543,Z 1055.941,A -85,B 0,C 180,E1 -29467.284,E2 -29467.284} C_VEL
LIN {X 0,Y 128.07,Z 1050.846,A -85,B 0,C 180,E1 -29478.423,E2 -29478.423} C_VEL
LIN {X 0,Y 141.11,Z 1045.148,A -85,B 0,C 180,E1 -29486.001,E2 -29486.001} C_VEL
LIN {X 0,Y 157.66,Z 1037.371,A -85,B 0,C 180,E1 -29492.83,E2 -29492.83} C_VEL
LIN {X 0,Y 174.66,Z 1028.309,A -85,B 0,C 180,E1 -29498.035,E2 -29498.035} C_VEL
LIN {X 0,Y 192.199,Z 1018.053,A -85,B 0,C 180,E1 -29502.182,E2 -29502.182} C_VEL
LIN {X 0,Y 211.107,Z 1005.519,A -85,B 0,C 180,E1 -29505.742,E2 -29505.742} C_VEL
LIN {X 0,Y 227.706,Z 993.281,A -85,B 0,C 180,E1 -29508.301,E2 -29508.301} C_VEL
LIN {X 0,Y 247.145,Z 977.121,A -85,B 0,C 180,E1 -29510.811,E2 -29510.811} C_VEL
LIN {X 0,Y 263.18,Z 962.114,A -85,B 0,C 180,E1 -29512.571,E2 -29512.571} C_VEL
LIN {X 0,Y 281.13,Z 943.115,A -85,B 0,C 180,E1 -29514.285,E2 -29514.285} C_VEL
LIN {X 0,Y 294.897,Z 926.623,A -85,B 0,C 180,E1 -29515.451,E2 -29515.451} C_VEL
LIN {X 0,Y 310.01,Z 906.158,A -85,B 0,C 180,E1 -29516.604,E2 -29516.604} C_VEL
LIN {X 0,Y 322.282,Z 887.027,A -85,B 0,C 180,E1 -29517.456,E2 -29517.456} C_VEL
LIN {X 0,Y 334.124,Z 866.025,A -85,B 0,C 180,E1 -29518.221,E2 -29518.221} C_VEL
LIN {X 0,Y 344.531,Z 844.055,A -85,B 0,C 180,E1 -29518.851,E2 -29518.851} C_VEL
LIN {X 0,Y 353.231,Z 822.577,A -85,B 0,C 180,E1 -29519.351,E2 -29519.351} C_VEL
LIN {X 0,Y 361.031,Z 798.65,A -85,B 0,C 180,E1 -29519.793,E2 -29519.793} C_VEL
LIN {X 0,Y 366.804,Z 776.382,A -85,B 0,C 180,E1 -29520.109,E2 -29520.109} C_VEL
LIN {X 0,Y 371.625,Z 750.591,A -85,B 0,C 180,E1 -29520.407,E2 -29520.407} C_VEL
LIN {X 0,Y 376.911,Z 709.347,A -85,B 0,C 180,E1 -29520.866,E2 -29520.866} C_VEL
LIN {X 0,Y 370.706,Z 756.915,A -85,B 0,C 180,E1 -29521.39,E2 -29521.39} C_VEL
LIN {X 0,Y 365.619,Z 781.495,A -85,B 0,C 180,E1 -29521.671,E2 -29521.671} C_VEL
LIN {X 0,Y 359.172,Z 805.343,A -85,B 0,C 180,E1 -29521.966,E2 -29521.966} C_VEL
LIN {X 0,Y 351.25,Z 828.005,A -85,B 0,C 180,E1 -29522.322,E2 -29522.322} C_VEL
LIN {X 0,Y 342.853,Z 848.262,A -85,B 0,C 180,E1 -29522.736,E2 -29522.736} C_VEL
LIN {X 0,Y 331.525,Z 871.314,A -85,B 0,C 180,E1 -29523.336,E2 -29523.336} C_VEL
LIN {X 0,Y 320.729,Z 890.198,A -85,B 0,C 180,E1 -29523.957,E2 -29523.957} C_VEL
LIN {X 0,Y 307.059,Z 911.202,A -85,B 0,C 180,E1 -29524.834,E2 -29524.834} C_VEL
LIN {X 0,Y 292.984,Z 929.939,A -85,B 0,C 180,E1 -29525.831,E2 -29525.831} C_VEL
LIN {X 0,Y 277.582,Z 948.286,A -85,B 0,C 180,E1 -29527.073,E2 -29527.073} C_VEL
LIN {X 0,Y 274.85,Z 951.224,A -85,B 0,C 180,E1 -29527.306,E2 -29527.306} C_VEL
LIN {X 0,Y 269.489,Z 956.787,A -85,B 0,C 180,E1 -29527.558,E2 -29527.558} C_VEL
LIN {X 0,Y 253.992,Z 971.309,A -85,B 0,C 180,E1 -29527.542,E2 -29527.542} C_VEL
LIN {X 0,Y 249.132,Z 975.586,A -85,B 0,C 180,E1 -29527.835,E2 -29527.835} C_VEL
LIN {X 0,Y 232.222,Z 990.065,A -85,B 0,C 180,E1 -29529.667,E2 -29529.667} C_VEL
LIN {X 0,Y 211.862,Z 1005.514,A -85,B 0,C 180,E1 -29532.327,E2 -29532.327} C_VEL
LIN {X 0,Y 194.686,Z 1017.099,A -85,B 0,C 180,E1 -29535.083,E2 -29535.083} C_VEL
LIN {X 0,Y 174.635,Z 1029.209,A -85,B 0,C 180,E1 -29539.139,E2 -29539.139} C_VEL
LIN {X 0,Y 157.259,Z 1038.502,A -85,B 0,C 180,E1 -29543.711,E2 -29543.711} C_VEL
LIN {X 0,Y 138.955,Z 1047.398,A -85,B 0,C 180,E1 -29550.245,E2 -29550.245} C_VEL
LIN {X 0,Y 123.418,Z 1054.125,A -85,B 0,C 180,E1 -29558.2,E2 -29558.2} C_VEL
LIN {X 0,Y 110.255,Z 1059.612,A -85,B 0,C 180,E1 -29568.545,E2 -29568.545} C_VEL
LIN {X 0,Y 101.103,Z 1063.279,A -85,B 0,C 180,E1 -29581.014,E2 -29581.014} C_VEL
LIN {X 0,Y 97.04,Z 1065.183,A -85,B 0,C 180,E1 -29592.614,E2 -29592.614} C_VEL
LIN {X 0,Y 96.007,Z 1065.973,A -85,B 0,C 180,E1 -29604.022,E2 -29604.022} C_VEL
LIN {X 0,Y 96.048,Z 1065.87,A -85,B 0,C 180,E1 -29611.79,E2 -29611.79} C_VEL
LIN {X 0,Y 96.117,Z 1065.222,A -85,B 0,C 180,E1 -29620.186,E2 -29620.186} C_VEL
LIN {X 0,Y 97.878,Z 1063.551,A -85,B 0,C 180,E1 -29630.95,E2 -29630.95} C_VEL
LIN {X 0,Y 103.223,Z 1060.462,A -85,B 0,C 180,E1 -29642.851,E2 -29642.851} C_VEL
LIN {X 0,Y 114.077,Z 1055.067,A -85,B 0,C 180,E1 -29655.232,E2 -29655.232} C_VEL
LIN {X 0,Y 126.363,Z 1049.078,A -85,B 0,C 180,E1 -29663.814,E2 -29663.814} C_VEL
LIN {X 0,Y 143.055,Z 1040.576,A -85,B 0,C 180,E1 -29671.725,E2 -29671.725} C_VEL
LIN {X 0,Y 159.38,Z 1031.449,A -85,B 0,C 180,E1 -29677.253,E2 -29677.253} C_VEL
LIN {X 0,Y 178.099,Z 1020.059,A -85,B 0,C 180,E1 -29682.014,E2 -29682.014} C_VEL
LIN {X 0,Y 196.16,Z 1007.623,A -85,B 0,C 180,E1 -29685.578,E2 -29685.578} C_VEL
LIN {X 0,Y 214.315,Z 993.867,A -85,B 0,C 180,E1 -29688.451,E2 -29688.451} C_VEL
LIN {X 0,Y 231.985,Z 978.69,A -85,B 0,C 180,E1 -29690.76,E2 -29690.76} C_VEL
LIN {X 0,Y 247.121,Z 964.299,A -85,B 0,C 180,E1 -29692.44,E2 -29692.44} C_VEL
LIN {X 0,Y 265.341,Z 944.789,A -85,B 0,C 180,E1 -29694.174,E2 -29694.174} C_VEL
LIN {X 0,Y 278.906,Z 928.369,A -85,B 0,C 180,E1 -29695.303,E2 -29695.303} C_VEL
LIN {X 0,Y 294.013,Z 907.779,A -85,B 0,C 180,E1 -29696.407,E2 -29696.407} C_VEL
LIN {X 0,Y 306.326,Z 888.461,A -85,B 0,C 180,E1 -29697.221,E2 -29697.221} C_VEL
LIN {X 0,Y 318.432,Z 866.87,A -85,B 0,C 180,E1 -29697.936,E2 -29697.936} C_VEL
LIN {X 0,Y 328.577,Z 845.349,A -85,B 0,C 180,E1 -29698.491,E2 -29698.491} C_VEL
LIN {X 0,Y 337.52,Z 823.187,A -85,B 0,C 180,E1 -29698.94,E2 -29698.94} C_VEL
LIN {X 0,Y 345.393,Z 798.893,A -85,B 0,C 180,E1 -29699.31,E2 -29699.31} C_VEL
LIN {X 0,Y 351.22,Z 776.228,A -85,B 0,C 180,E1 -29699.588,E2 -29699.588} C_VEL
LIN {X 0,Y 355.924,Z 750.691,A -85,B 0,C 180,E1 -29699.882,E2 -29699.882} C_VEL
LIN {X 0,Y 365.441,Z 674.378,A -85,B 0,C 180,E1 -29700.732,E2 -29700.732} C_VEL
LIN {X 0,Y 365.453,Z 674.197,A -85,B 0,C 180,E1 -29701.411,E2 -29701.411} C_VEL
LIN {X 0,Y 365.423,Z 674.503,A -85,B 0,C 180,E1 -29701.643,E2 -29701.643} C_VEL
LIN {X 0,Y 355.505,Z 753.47,A -85,B 0,C 180,E1 -29702.51,E2 -29702.51} C_VEL
LIN {X 0,Y 350.522,Z 778.873,A -85,B 0,C 180,E1 -29702.816,E2 -29702.816} C_VEL
LIN {X 0,Y 344.791,Z 800.65,A -85,B 0,C 180,E1 -29703.139,E2 -29703.139} C_VEL
LIN {X 0,Y 336.631,Z 825.054,A -85,B 0,C 180,E1 -29703.61,E2 -29703.61} C_VEL
LIN {X 0,Y 328.294,Z 845.491,A -85,B 0,C 180,E1 -29704.114,E2 -29704.114} C_VEL
LIN {X 0,Y 317.524,Z 867.951,A -85,B 0,C 180,E1 -29704.797,E2 -29704.797} C_VEL
LIN {X 0,Y 305.914,Z 888.421,A -85,B 0,C 180,E1 -29705.577,E2 -29705.577} C_VEL
LIN {X 0,Y 292.385,Z 909.331,A -85,B 0,C 180,E1 -29706.565,E2 -29706.565} C_VEL
LIN {X 0,Y 277.993,Z 928.505,A -85,B 0,C 180,E1 -29707.727,E2 -29707.727} C_VEL
LIN {X 0,Y 262.306,Z 947.137,A -85,B 0,C 180,E1 -29709.146,E2 -29709.146} C_VEL
LIN {X 0,Y 245.389,Z 964.604,A -85,B 0,C 180,E1 -29710.886,E2 -29710.886} C_VEL
LIN {X 0,Y 227.81,Z 980.892,A -85,B 0,C 180,E1 -29712.996,E2 -29712.996} C_VEL
LIN {X 0,Y 209.677,Z 995.591,A -85,B 0,C 180,E1 -29715.575,E2 -29715.575} C_VEL
LIN {X 0,Y 191.171,Z 1009.129,A -85,B 0,C 180,E1 -29718.793,E2 -29718.793} C_VEL
LIN {X 0,Y 172.586,Z 1021.044,A -85,B 0,C 180,E1 -29722.841,E2 -29722.841} C_VEL
LIN {X 0,Y 154.901,Z 1031.369,A -85,B 0,C 180,E1 -29727.83,E2 -29727.83} C_VEL
LIN {X 0,Y 137.923,Z 1040.139,A -85,B 0,C 180,E1 -29734.264,E2 -29734.264} C_VEL
LIN {X 0,Y 122.978,Z 1047.366,A -85,B 0,C 180,E1 -29742.278,E2 -29742.278} C_VEL
LIN {X 0,Y 110.299,Z 1053.09,A -85,B 0,C 180,E1 -29752.601,E2 -29752.601} C_VEL
LIN {X 0,Y 102.317,Z 1056.798,A -85,B 0,C 180,E1 -29763.286,E2 -29763.286} C_VEL
LIN {X 0,Y 97.271,Z 1059.603,A -85,B 0,C 180,E1 -29776.93,E2 -29776.93} C_VEL
LIN {X 0,Y 96.111,Z 1060.667,A -85,B 0,C 180,E1 -29788.212,E2 -29788.212} C_VEL
LIN {X 0,Y 96.193,Z 1060.888,A -85,B 0,C 180,E1 -29797.766,E2 -29797.766} C_VEL
LIN {X 0,Y 97.763,Z 1060.262,A -85,B 0,C 180,E1 -29809.104,E2 -29809.104} C_VEL
LIN {X 0,Y 102.316,Z 1058.578,A -85,B 0,C 180,E1 -29820.542,E2 -29820.542} C_VEL
LIN {X 0,Y 111.891,Z 1055.195,A -85,B 0,C 180,E1 -29832.778,E2 -29832.778} C_VEL
LIN {X 0,Y 125.302,Z 1049.99,A -85,B 0,C 180,E1 -29842.938,E2 -29842.938} C_VEL
LIN {X 0,Y 141.681,Z 1043.231,A -85,B 0,C 180,E1 -29851.058,E2 -29851.058} C_VEL
LIN {X 0,Y 159.386,Z 1034.846,A -85,B 0,C 180,E1 -29857.248,E2 -29857.248} C_VEL
LIN {X 0,Y 177.673,Z 1025.286,A -85,B 0,C 180,E1 -29862.004,E2 -29862.004} C_VEL
LIN {X 0,Y 196.95,Z 1013.725,A -85,B 0,C 180,E1 -29865.895,E2 -29865.895} C_VEL
LIN {X 0,Y 215.062,Z 1001.627,A -85,B 0,C 180,E1 -29868.814,E2 -29868.814} C_VEL
LIN {X 0,Y 233.668,Z 987.512,A -85,B 0,C 180,E1 -29871.293,E2 -29871.293} C_VEL
LIN {X 0,Y 249.776,Z 973.849,A -85,B 0,C 180,E1 -29873.112,E2 -29873.112} C_VEL
LIN {X 0,Y 268.521,Z 955.929,A -85,B 0,C 180,E1 -29874.931,E2 -29874.931} C_VEL
LIN {X 0,Y 283.591,Z 939.584,A -85,B 0,C 180,E1 -29876.205,E2 -29876.205} C_VEL
LIN {X 0,Y 299.769,Z 919.763,A -85,B 0,C 180,E1 -29877.428,E2 -29877.428} C_VEL
LIN {X 0,Y 312.603,Z 901.752,A -85,B 0,C 180,E1 -29878.301,E2 -29878.301} C_VEL
LIN {X 0,Y 325.766,Z 880.868,A -85,B 0,C 180,E1 -29879.121,E2 -29879.121} C_VEL
LIN {X 0,Y 336.965,Z 859.912,A -85,B 0,C 180,E1 -29879.786,E2 -29879.786} C_VEL
LIN {X 0,Y 346.968,Z 838.28,A -85,B 0,C 180,E1 -29880.332,E2 -29880.332} C_VEL
LIN {X 0,Y 355.745,Z 815.19,A -85,B 0,C 180,E1 -29880.791,E2 -29880.791} C_VEL
LIN {X 0,Y 355.996,Z 814.447,A -85,B 0,C 180,E1 -29880.812,E2 -29880.812} C_VEL
LIN {X 0,Y 347.584,Z 836.962,A -85,B 0,C 180,E1 -29881.169,E2 -29881.169} C_VEL
LIN {X 0,Y 337.598,Z 858.809,A -85,B 0,C 180,E1 -29881.621,E2 -29881.621} C_VEL
LIN {X 0,Y 326.699,Z 879.453,A -85,B 0,C 180,E1 -29882.174,E2 -29882.174} C_VEL
LIN {X 0,Y 313.371,Z 901.034,A -85,B 0,C 180,E1 -29882.913,E2 -29882.913} C_VEL
LIN {X 0,Y 300.592,Z 919.194,A -85,B 0,C 180,E1 -29883.697,E2 -29883.697} C_VEL
LIN {X 0,Y 283.805,Z 940.086,A -85,B 0,C 180,E1 -29884.85,E2 -29884.85} C_VEL
LIN {X 0,Y 268.954,Z 956.383,A -85,B 0,C 180,E1 -29886.021,E2 -29886.021} C_VEL
LIN {X 0,Y 250.243,Z 974.596,A -85,B 0,C 180,E1 -29887.724,E2 -29887.724} C_VEL
LIN {X 0,Y 249.132,Z 975.586,A -85,B 0,C 180,E1 -29887.835,E2 -29887.835} C_VEL
LIN {X 0,Y 243.334,Z 980.64,A -85,B 0,C 180,E1 -29888.176,E2 -29888.176} C_VEL
LIN {X 0,Y 226.542,Z 993.597,A -85,B 0,C 180,E1 -29888.354,E2 -29888.354} C_VEL
LIN {X 0,Y 221.349,Z 997.367,A -85,B 0,C 180,E1 -29888.746,E2 -29888.746} C_VEL
LIN {X 0,Y 202.819,Z 1010.504,A -85,B 0,C 180,E1 -29891.168,E2 -29891.168} C_VEL
LIN {X 0,Y 182.748,Z 1022.98,A -85,B 0,C 180,E1 -29894.433,E2 -29894.433} C_VEL
LIN {X 0,Y 165.138,Z 1032.771,A -85,B 0,C 180,E1 -29898.082,E2 -29898.082} C_VEL
LIN {X 0,Y 144.307,Z 1042.999,A -85,B 0,C 180,E1 -29903.849,E2 -29903.849} C_VEL
LIN {X 0,Y 127.501,Z 1050.331,A -85,B 0,C 180,E1 -29910.385,E2 -29910.385} C_VEL
LIN {X 0,Y 110.313,Z 1057.079,A -85,B 0,C 180,E1 -29920.414,E2 -29920.414} C_VEL
LIN {X 0,Y 98.962,Z 1061.257,A -85,B 0,C 180,E1 -29931.212,E2 -29931.212} C_VEL
LIN {X 0,Y 90.63,Z 1064.429,A -85,B 0,C 180,E1 -29946.307,E2 -29946.307} C_VEL
LIN {X 0,Y 88.134,Z 1065.603,A -85,B 0,C 180,E1 -29959.542,E2 -29959.542} C_VEL
LIN {X 0,Y 88.052,Z 1065.765,A -85,B 0,C 180,E1 -29968.699,E2 -29968.699} C_VEL
LIN {X 0,Y 88.023,Z 1065.425,A -85,B 0,C 180,E1 -29977.178,E2 -29977.178} C_VEL
LIN {X 0,Y 89.748,Z 1063.674,A -85,B 0,C 180,E1 -29990.886,E2 -29990.886} C_VEL
LIN {X 0,Y 95.301,Z 1060.719,A -85,B 0,C 180,E1 -30003.784,E2 -30003.784} C_VEL
LIN {X 0,Y 106.474,Z 1055.721,A -85,B 0,C 180,E1 -30016.722,E2 -30016.722} C_VEL
LIN {X 0,Y 120.287,Z 1049.437,A -85,B 0,C 180,E1 -30026.227,E2 -30026.227} C_VEL
LIN {X 0,Y 136.984,Z 1041.509,A -85,B 0,C 180,E1 -30033.872,E2 -30033.872} C_VEL
LIN {X 0,Y 155.517,Z 1031.63,A -85,B 0,C 180,E1 -30039.834,E2 -30039.834} C_VEL
LIN {X 0,Y 173.581,Z 1021.061,A -85,B 0,C 180,E1 -30044.15,E2 -30044.15} C_VEL
LIN {X 0,Y 192.966,Z 1008.226,A -85,B 0,C 180,E1 -30047.734,E2 -30047.734} C_VEL
LIN {X 0,Y 210.003,Z 995.679,A -85,B 0,C 180,E1 -30050.262,E2 -30050.262} C_VEL
LIN {X 0,Y 229.85,Z 979.204,A -85,B 0,C 180,E1 -30052.676,E2 -30052.676} C_VEL
LIN {X 0,Y 246.174,Z 963.947,A -85,B 0,C 180,E1 -30054.337,E2 -30054.337} C_VEL
LIN {X 0,Y 263.748,Z 945.429,A -85,B 0,C 180,E1 -30055.869,E2 -30055.869} C_VEL
LIN {X 0,Y 277.864,Z 928.591,A -85,B 0,C 180,E1 -30056.946,E2 -30056.946} C_VEL
LIN {X 0,Y 292.658,Z 908.786,A -85,B 0,C 180,E1 -30057.934,E2 -30057.934} C_VEL
LIN {X 0,Y 305.543,Z 888.83,A -85,B 0,C 180,E1 -30058.714,E2 -30058.714} C_VEL
LIN {X 0,Y 317.485,Z 867.823,A -85,B 0,C 180,E1 -30059.358,E2 -30059.358} C_VEL
LIN {X 0,Y 327.964,Z 845.95,A -85,B 0,C 180,E1 -30059.879,E2 -30059.879} C_VEL
LIN {X 0,Y 336.413,Z 825.329,A -85,B 0,C 180,E1 -30060.268,E2 -30060.268} C_VEL
LIN {X 0,Y 344.92,Z 799.821,A -85,B 0,C 180,E1 -30060.629,E2 -30060.629} C_VEL
LIN {X 0,Y 350.662,Z 777.897,A -85,B 0,C 180,E1 -30060.877,E2 -30060.877} C_VEL
LIN {X 0,Y 355.751,Z 751.195,A -85,B 0,C 180,E1 -30061.168,E2 -30061.168} C_VEL
LIN {X 0,Y 355.896,Z 750.203,A -85,B 0,C 180,E1 -30061.183,E2 -30061.183} C_VEL
LIN {X 0,Y 351.231,Z 775.465,A -85,B 0,C 180,E1 -30061.46,E2 -30061.46} C_VEL
LIN {X 0,Y 345.359,Z 798.186,A -85,B 0,C 180,E1 -30061.766,E2 -30061.766} C_VEL
LIN {X 0,Y 337.706,Z 821.81,A -85,B 0,C 180,E1 -30062.178,E2 -30062.178} C_VEL
LIN {X 0,Y 328.819,Z 843.752,A -85,B 0,C 180,E1 -30062.665,E2 -30062.665} C_VEL
LIN {X 0,Y 318.916,Z 864.668,A -85,B 0,C 180,E1 -30063.235,E2 -30063.235} C_VEL
LIN {X 0,Y 306.707,Z 886.457,A -85,B 0,C 180,E1 -30063.985,E2 -30063.985} C_VEL
LIN {X 0,Y 294.496,Z 905.464,A -85,B 0,C 180,E1 -30064.79,E2 -30064.79} C_VEL
LIN {X 0,Y 278.96,Z 926.488,A -85,B 0,C 180,E1 -30065.926,E2 -30065.926} C_VEL
LIN {X 0,Y 264.982,Z 943.141,A -85,B 0,C 180,E1 -30067.064,E2 -30067.064} C_VEL
LIN {X 0,Y 246.837,Z 962.211,A -85,B 0,C 180,E1 -30068.736,E2 -30068.736} C_VEL
LIN {X 0,Y 231.737,Z 976.253,A -85,B 0,C 180,E1 -30070.339,E2 -30070.339} C_VEL
LIN {X 0,Y 213.152,Z 991.768,A -85,B 0,C 180,E1 -30072.652,E2 -30072.652} C_VEL
LIN {X 0,Y 194.957,Z 1005.081,A -85,B 0,C 180,E1 -30075.376,E2 -30075.376} C_VEL
LIN {X 0,Y 176.117,Z 1017.5,A -85,B 0,C 180,E1 -30078.882,E2 -30078.882} C_VEL
LIN {X 0,Y 157.776,Z 1028.058,A -85,B 0,C 180,E1 -30083.231,E2 -30083.231} C_VEL
LIN {X 0,Y 140.261,Z 1037.215,A -85,B 0,C 180,E1 -30088.736,E2 -30088.736} C_VEL
LIN {X 0,Y 122.904,Z 1045.263,A -85,B 0,C 180,E1 -30096.349,E2 -30096.349} C_VEL
LIN {X 0,Y 109.249,Z 1051.162,A -85,B 0,C 180,E1 -30105.192,E2 -30105.192} C_VEL
LIN {X 0,Y 97.328,Z 1056.113,A -85,B 0,C 180,E1 -30117.709,E2 -30117.709} C_VEL
LIN {X 0,Y 91.023,Z 1058.925,A -85,B 0,C 180,E1 -30130.091,E2 -30130.091} C_VEL
LIN {X 0,Y 88.453,Z 1060.477,A -85,B 0,C 180,E1 -30142.204,E2 -30142.204} C_VEL
LIN {X 0,Y 88.054,Z 1061.026,A -85,B 0,C 180,E1 -30152.165,E2 -30152.165} C_VEL
LIN {X 0,Y 88.473,Z 1061.001,A -85,B 0,C 180,E1 -30161.738,E2 -30161.738} C_VEL
LIN {X 0,Y 91.091,Z 1060.152,A -85,B 0,C 180,E1 -30173.963,E2 -30173.963} C_VEL
LIN {X 0,Y 99.237,Z 1057.566,A -85,B 0,C 180,E1 -30188.66,E2 -30188.66} C_VEL
LIN {X 0,Y 110.436,Z 1053.779,A -85,B 0,C 180,E1 -30199.512,E2 -30199.512} C_VEL
LIN {X 0,Y 126.018,Z 1048.173,A -85,B 0,C 180,E1 -30208.974,E2 -30208.974} C_VEL
LIN {X 0,Y 143.827,Z 1040.75,A -85,B 0,C 180,E1 -30216.22,E2 -30216.22} C_VEL
LIN {X 0,Y 163.131,Z 1031.79,A -85,B 0,C 180,E1 -30221.815,E2 -30221.815} C_VEL
LIN {X 0,Y 182.729,Z 1021.212,A -85,B 0,C 180,E1 -30226.068,E2 -30226.068} C_VEL
LIN {X 0,Y 202.435,Z 1009.317,A -85,B 0,C 180,E1 -30229.396,E2 -30229.396} C_VEL
LIN {X 0,Y 221.152,Z 996.301,A -85,B 0,C 180,E1 -30231.956,E2 -30231.956} C_VEL
LIN {X 0,Y 239.277,Z 982.251,A -85,B 0,C 180,E1 -30234.016,E2 -30234.016} C_VEL
LIN {X 0,Y 257.666,Z 965.973,A -85,B 0,C 180,E1 -30235.794,E2 -30235.794} C_VEL
LIN {X 0,Y 273.319,Z 950.438,A -85,B 0,C 180,E1 -30237.106,E2 -30237.106} C_VEL
LIN {X 0,Y 290.584,Z 930.957,A -85,B 0,C 180,E1 -30238.383,E2 -30238.383} C_VEL
LIN {X 0,Y 303.991,Z 913.78,A -85,B 0,C 180,E1 -30239.275,E2 -30239.275} C_VEL
LIN {X 0,Y 318.966,Z 891.862,A -85,B 0,C 180,E1 -30240.172,E2 -30240.172} C_VEL
LIN {X 0,Y 328.112,Z 876.569,A -85,B 0,C 180,E1 -30240.681,E2 -30240.681} C_VEL
LIN {X 0,Y 314.057,Z 899.556,A -85,B 0,C 180,E1 -30241.382,E2 -30241.382} C_VEL
LIN {X 0,Y 301.168,Z 917.831,A -85,B 0,C 180,E1 -30242.093,E2 -30242.093} C_VEL
LIN {X 0,Y 284.882,Z 938.162,A -85,B 0,C 180,E1 -30243.1,E2 -30243.1} C_VEL
LIN {X 0,Y 269.198,Z 955.294,A -85,B 0,C 180,E1 -30244.213,E2 -30244.213} C_VEL
LIN {X 0,Y 251.21,Z 972.801,A -85,B 0,C 180,E1 -30245.689,E2 -30245.689} C_VEL
LIN {X 0,Y 233.664,Z 987.783,A -85,B 0,C 180,E1 -30247.376,E2 -30247.376} C_VEL
LIN {X 0,Y 221.349,Z 997.367,A -85,B 0,C 180,E1 -30248.746,E2 -30248.746} C_VEL
LIN {X 0,Y 215.178,Z 1001.856,A -85,B 0,C 180,E1 -30249.21,E2 -30249.21} C_VEL
LIN {X 0,Y 197.259,Z 1013.111,A -85,B 0,C 180,E1 -30249.653,E2 -30249.653} C_VEL
LIN {X 0,Y 191.798,Z 1016.364,A -85,B 0,C 180,E1 -30250.185,E2 -30250.185} C_VEL
LIN {X 0,Y 170.831,Z 1028.435,A -85,B 0,C 180,E1 -30253.685,E2 -30253.685} C_VEL
LIN {X 0,Y 152.223,Z 1037.766,A -85,B 0,C 180,E1 -30257.741,E2 -30257.741} C_VEL
LIN {X 0,Y 132.598,Z 1046.572,A -85,B 0,C 180,E1 -30263.557,E2 -30263.557} C_VEL
LIN {X 0,Y 114.639,Z 1053.495,A -85,B 0,C 180,E1 -30271.266,E2 -30271.266} C_VEL
LIN {X 0,Y 99.066,Z 1059.019,A -85,B 0,C 180,E1 -30281.678,E2 -30281.678} C_VEL
LIN {X 0,Y 87.485,Z 1062.753,A -85,B 0,C 180,E1 -30295.147,E2 -30295.147} C_VEL
LIN {X 0,Y 81.821,Z 1064.694,A -85,B 0,C 180,E1 -30308.493,E2 -30308.493} C_VEL
LIN {X 0,Y 80.039,Z 1065.524,A -85,B 0,C 180,E1 -30322.101,E2 -30322.101} C_VEL
LIN {X 0,Y 80.065,Z 1065.483,A -85,B 0,C 180,E1 -30330.715,E2 -30330.715} C_VEL
LIN {X 0,Y 80.143,Z 1064.915,A -85,B 0,C 180,E1 -30340.786,E2 -30340.786} C_VEL
LIN {X 0,Y 82.601,Z 1063.202,A -85,B 0,C 180,E1 -30354.304,E2 -30354.304} C_VEL
LIN {X 0,Y 89.405,Z 1060.143,A -85,B 0,C 180,E1 -30367.96,E2 -30367.96} C_VEL
LIN {X 0,Y 103.092,Z 1054.553,A -85,B 0,C 180,E1 -30381.778,E2 -30381.778} C_VEL
LIN {X 0,Y 117.353,Z 1048.538,A -85,B 0,C 180,E1 -30390.384,E2 -30390.384} C_VEL
LIN {X 0,Y 136.792,Z 1039.602,A -85,B 0,C 180,E1 -30398.173,E2 -30398.173} C_VEL
LIN {X 0,Y 154.592,Z 1030.405,A -85,B 0,C 180,E1 -30403.187,E2 -30403.187} C_VEL
LIN {X 0,Y 175.138,Z 1018.524,A -85,B 0,C 180,E1 -30407.491,E2 -30407.491} C_VEL
LIN {X 0,Y 192.704,Z 1006.997,A -85,B 0,C 180,E1 -30410.353,E2 -30410.353} C_VEL
LIN {X 0,Y 211.627,Z 993.223,A -85,B 0,C 180,E1 -30412.84,E2 -30412.84} C_VEL
LIN {X 0,Y 229.914,Z 978.005,A -85,B 0,C 180,E1 -30414.82,E2 -30414.82} C_VEL
LIN {X 0,Y 246.479,Z 962.656,A -85,B 0,C 180,E1 -30416.328,E2 -30416.328} C_VEL
LIN {X 0,Y 264.181,Z 944.031,A -85,B 0,C 180,E1 -30417.715,E2 -30417.715} C_VEL
LIN {X 0,Y 278.388,Z 927.159,A -85,B 0,C 180,E1 -30418.685,E2 -30418.685} C_VEL
LIN {X 0,Y 294.473,Z 905.391,A -85,B 0,C 180,E1 -30419.645,E2 -30419.645} C_VEL
LIN {X 0,Y 306.513,Z 886.674,A -85,B 0,C 180,E1 -30420.295,E2 -30420.295} C_VEL
LIN {X 0,Y 319.052,Z 864.267,A -85,B 0,C 180,E1 -30420.898,E2 -30420.898} C_VEL
LIN {X 0,Y 328.048,Z 845.409,A -85,B 0,C 180,E1 -30421.298,E2 -30421.298} C_VEL
LIN {X 0,Y 317.135,Z 867.907,A -85,B 0,C 180,E1 -30421.877,E2 -30421.877} C_VEL
LIN {X 0,Y 305.267,Z 888.511,A -85,B 0,C 180,E1 -30422.545,E2 -30422.545} C_VEL
LIN {X 0,Y 291.969,Z 908.796,A -85,B 0,C 180,E1 -30423.356,E2 -30423.356} C_VEL
LIN {X 0,Y 277.285,Z 928.057,A -85,B 0,C 180,E1 -30424.343,E2 -30424.343} C_VEL
LIN {X 0,Y 262.321,Z 945.54,A -85,B 0,C 180,E1 -30425.468,E2 -30425.468} C_VEL
LIN {X 0,Y 244.776,Z 963.475,A -85,B 0,C 180,E1 -30426.958,E2 -30426.958} C_VEL
LIN {X 0,Y 228.518,Z 978.259,A -85,B 0,C 180,E1 -30428.556,E2 -30428.556} C_VEL
LIN {X 0,Y 208.712,Z 994.157,A -85,B 0,C 180,E1 -30430.855,E2 -30430.855} C_VEL
LIN {X 0,Y 191.334,Z 1006.498,A -85,B 0,C 180,E1 -30433.294,E2 -30433.294} C_VEL
LIN {X 0,Y 170.399,Z 1019.643,A -85,B 0,C 180,E1 -30436.967,E2 -30436.967} C_VEL
LIN {X 0,Y 153.038,Z 1029.242,A -85,B 0,C 180,E1 -30440.884,E2 -30440.884} C_VEL
LIN {X 0,Y 133.346,Z 1038.953,A -85,B 0,C 180,E1 -30446.834,E2 -30446.834} C_VEL
LIN {X 0,Y 116.827,Z 1046.116,A -85,B 0,C 180,E1 -30453.882,E2 -30453.882} C_VEL
LIN {X 0,Y 101.262,Z 1052.384,A -85,B 0,C 180,E1 -30463.878,E2 -30463.878} C_VEL
LIN {X 0,Y 89.323,Z 1056.815,A -85,B 0,C 180,E1 -30476.735,E2 -30476.735} C_VEL
LIN {X 0,Y 82.695,Z 1059.54,A -85,B 0,C 180,E1 -30490.583,E2 -30490.583} C_VEL
LIN {X 0,Y 80.2,Z 1061.036,A -85,B 0,C 180,E1 -30505.71,E2 -30505.71} C_VEL
LIN {X 0,Y 80.106,Z 1061.354,A -85,B 0,C 180,E1 -30515.731,E2 -30515.731} C_VEL
LIN {X 0,Y 81.637,Z 1060.995,A -85,B 0,C 180,E1 -30529.311,E2 -30529.311} C_VEL
LIN {X 0,Y 87.429,Z 1059.308,A -85,B 0,C 180,E1 -30544.083,E2 -30544.083} C_VEL
LIN {X 0,Y 97.026,Z 1056.529,A -85,B 0,C 180,E1 -30556.169,E2 -30556.169} C_VEL
LIN {X 0,Y 113.467,Z 1051.27,A -85,B 0,C 180,E1 -30568.08,E2 -30568.08} C_VEL
LIN {X 0,Y 129.65,Z 1045.379,A -85,B 0,C 180,E1 -30575.512,E2 -30575.512} C_VEL
LIN {X 0,Y 150.284,Z 1036.767,A -85,B 0,C 180,E1 -30582.069,E2 -30582.069} C_VEL
LIN {X 0,Y 168.755,Z 1027.861,A -85,B 0,C 180,E1 -30586.34,E2 -30586.34} C_VEL
LIN {X 0,Y 189.82,Z 1016.29,A -85,B 0,C 180,E1 -30590.075,E2 -30590.075} C_VEL
LIN {X 0,Y 208.661,Z 1004.403,A -85,B 0,C 180,E1 -30592.715,E2 -30592.715} C_VEL
LIN {X 0,Y 228.838,Z 990.026,A -85,B 0,C 180,E1 -30595.021,E2 -30595.021} C_VEL
LIN {X 0,Y 246.38,Z 975.724,A -85,B 0,C 180,E1 -30596.706,E2 -30596.706} C_VEL
LIN {X 0,Y 264.601,Z 959.103,A -85,B 0,C 180,E1 -30598.2,E2 -30598.2} C_VEL
LIN {X 0,Y 281.179,Z 941.699,A -85,B 0,C 180,E1 -30599.389,E2 -30599.389} C_VEL
LIN {X 0,Y 296.878,Z 923.215,A -85,B 0,C 180,E1 -30600.386,E2 -30600.386} C_VEL
LIN {X 0,Y 300.211,Z 918.838,A -85,B 0,C 180,E1 -30600.589,E2 -30600.589} C_VEL
LIN {X 0,Y 283.073,Z 939.768,A -85,B 0,C 180,E1 -30601.553,E2 -30601.553} C_VEL
LIN {X 0,Y 268.228,Z 955.73,A -85,B 0,C 180,E1 -30602.512,E2 -30602.512} C_VEL
LIN {X 0,Y 249.527,Z 973.574,A -85,B 0,C 180,E1 -30603.906,E2 -30603.906} C_VEL
LIN {X 0,Y 232.02,Z 988.26,A -85,B 0,C 180,E1 -30605.441,E2 -30605.441} C_VEL
LIN {X 0,Y 212.779,Z 1002.699,A -85,B 0,C 180,E1 -30607.463,E2 -30607.463} C_VEL
LIN {X 0,Y 192.923,Z 1015.667,A -85,B 0,C 180,E1 -30610.022,E2 -30610.022} C_VEL
LIN {X 0,Y 191.798,Z 1016.364,A -85,B 0,C 180,E1 -30610.185,E2 -30610.185} C_VEL
LIN {X 0,Y 185.332,Z 1020.187,A -85,B 0,C 180,E1 -30610.825,E2 -30610.825} C_VEL
LIN {X 0,Y 167.501,Z 1029.198,A -85,B 0,C 180,E1 -30611.611,E2 -30611.611} C_VEL
LIN {X 0,Y 160.881,Z 1032.406,A -85,B 0,C 180,E1 -30612.444,E2 -30612.444} C_VEL
LIN {X 0,Y 139.306,Z 1042.3,A -85,B 0,C 180,E1 -30617.326,E2 -30617.326} C_VEL
LIN {X 0,Y 121.592,Z 1049.357,A -85,B 0,C 180,E1 -30622.926,E2 -30622.926} C_VEL
LIN {X 0,Y 102.483,Z 1056.058,A -85,B 0,C 180,E1 -30631.915,E2 -30631.915} C_VEL
LIN {X 0,Y 87.831,Z 1060.53,A -85,B 0,C 180,E1 -30643.231,E2 -30643.231} C_VEL
LIN {X 0,Y 76.857,Z 1063.792,A -85,B 0,C 180,E1 -30659.165,E2 -30659.165} C_VEL
LIN {X 0,Y 72.357,Z 1065.15,A -85,B 0,C 180,E1 -30676.413,E2 -30676.413} C_VEL
LIN {X 0,Y 72.042,Z 1065.346,A -85,B 0,C 180,E1 -30687.879,E2 -30687.879} C_VEL
LIN {X 0,Y 72.025,Z 1065.072,A -85,B 0,C 180,E1 -30697.177,E2 -30697.177} C_VEL
LIN {X 0,Y 74.261,Z 1063.444,A -85,B 0,C 180,E1 -30713.824,E2 -30713.824} C_VEL
LIN {X 0,Y 81.233,Z 1060.567,A -85,B 0,C 180,E1 -30728.884,E2 -30728.884} C_VEL
LIN {X 0,Y 93.633,Z 1056.048,A -85,B 0,C 180,E1 -30742.207,E2 -30742.207} C_VEL
LIN {X 0,Y 110.388,Z 1049.53,A -85,B 0,C 180,E1 -30752.583,E2 -30752.583} C_VEL
LIN {X 0,Y 127.162,Z 1042.412,A -85,B 0,C 180,E1 -30759.343,E2 -30759.343} C_VEL
LIN {X 0,Y 147.917,Z 1032.458,A -85,B 0,C 180,E1 -30765.162,E2 -30765.162} C_VEL
LIN {X 0,Y 166.091,Z 1022.567,A -85,B 0,C 180,E1 -30768.896,E2 -30768.896} C_VEL
LIN {X 0,Y 186.728,Z 1009.912,A -85,B 0,C 180,E1 -30772.153,E2 -30772.153} C_VEL
LIN {X 0,Y 204.943,Z 997.17,A -85,B 0,C 180,E1 -30774.437,E2 -30774.437} C_VEL
LIN {X 0,Y 224.412,Z 981.948,A -85,B 0,C 180,E1 -30776.425,E2 -30776.425} C_VEL
LIN {X 0,Y 242.13,Z 966.054,A -85,B 0,C 180,E1 -30777.937,E2 -30777.937} C_VEL
LIN {X 0,Y 258.999,Z 949.173,A -85,B 0,C 180,E1 -30779.163,E2 -30779.163} C_VEL
LIN {X 0,Y 275.526,Z 930.197,A -85,B 0,C 180,E1 -30780.208,E2 -30780.208} C_VEL
LIN {X 0,Y 290.012,Z 911.432,A -85,B 0,C 180,E1 -30781,E2 -30781} C_VEL
LIN {X 0,Y 298.058,Z 899.767,A -85,B 0,C 180,E1 -30781.417,E2 -30781.417} C_VEL
LIN {X 0,Y 285.17,Z 917.82,A -85,B 0,C 180,E1 -30782.157,E2 -30782.157} C_VEL
LIN {X 0,Y 268.398,Z 938.404,A -85,B 0,C 180,E1 -30783.237,E2 -30783.237} C_VEL
LIN {X 0,Y 253.642,Z 954.276,A -85,B 0,C 180,E1 -30784.296,E2 -30784.296} C_VEL
LIN {X 0,Y 236.156,Z 971.092,A -85,B 0,C 180,E1 -30785.735,E2 -30785.735} C_VEL
LIN {X 0,Y 217.834,Z 986.434,A -85,B 0,C 180,E1 -30787.49,E2 -30787.49} C_VEL
LIN {X 0,Y 198.809,Z 1000.684,A -85,B 0,C 180,E1 -30789.68,E2 -30789.68} C_VEL
LIN {X 0,Y 179.193,Z 1013.415,A -85,B 0,C 180,E1 -30792.449,E2 -30792.449} C_VEL
LIN {X 0,Y 160.082,Z 1024.484,A -85,B 0,C 180,E1 -30795.867,E2 -30795.867} C_VEL
LIN {X 0,Y 139.935,Z 1034.598,A -85,B 0,C 180,E1 -30800.602,E2 -30800.602} C_VEL
LIN {X 0,Y 121.77,Z 1042.674,A -85,B 0,C 180,E1 -30806.488,E2 -30806.488} C_VEL
LIN {X 0,Y 103.085,Z 1049.94,A -85,B 0,C 180,E1 -30815.436,E2 -30815.436} C_VEL
LIN {X 0,Y 89.246,Z 1054.832,A -85,B 0,C 180,E1 -30826.002,E2 -30826.002} C_VEL
LIN {X 0,Y 77.576,Z 1058.844,A -85,B 0,C 180,E1 -30842.354,E2 -30842.354} C_VEL
LIN {X 0,Y 73.023,Z 1060.664,A -85,B 0,C 180,E1 -30857.345,E2 -30857.345} C_VEL
LIN {X 0,Y 72.103,Z 1061.361,A -85,B 0,C 180,E1 -30869.206,E2 -30869.206} C_VEL
LIN {X 0,Y 72.33,Z 1061.523,A -85,B 0,C 180,E1 -30880.353,E2 -30880.353} C_VEL
LIN {X 0,Y 75.099,Z 1060.884,A -85,B 0,C 180,E1 -30895.218,E2 -30895.218} C_VEL
LIN {X 0,Y 82.063,Z 1059.185,A -85,B 0,C 180,E1 -30909.315,E2 -30909.315} C_VEL
LIN {X 0,Y 95.205,Z 1055.765,A -85,B 0,C 180,E1 -30922.958,E2 -30922.958} C_VEL
LIN {X 0,Y 111.334,Z 1050.788,A -85,B 0,C 180,E1 -30932.763,E2 -30932.763} C_VEL
LIN {X 0,Y 129.769,Z 1044.367,A -85,B 0,C 180,E1 -30940.056,E2 -30940.056} C_VEL
LIN {X 0,Y 149.722,Z 1036.129,A -85,B 0,C 180,E1 -30945.548,E2 -30945.548} C_VEL
LIN {X 0,Y 168.842,Z 1027.108,A -85,B 0,C 180,E1 -30949.438,E2 -30949.438} C_VEL
LIN {X 0,Y 190.474,Z 1015.29,A -85,B 0,C 180,E1 -30952.817,E2 -30952.817} C_VEL
LIN {X 0,Y 208.745,Z 1003.9,A -85,B 0,C 180,E1 -30955.083,E2 -30955.083} C_VEL
LIN {X 0,Y 230.237,Z 988.599,A -85,B 0,C 180,E1 -30957.263,E2 -30957.263} C_VEL
LIN {X 0,Y 247.037,Z 974.977,A -85,B 0,C 180,E1 -30958.693,E2 -30958.693} C_VEL
LIN {X 0,Y 265.971,Z 957.657,A -85,B 0,C 180,E1 -30960.078,E2 -30960.078} C_VEL
LIN {X 0,Y 272.432,Z 951.134,A -85,B 0,C 180,E1 -30960.502,E2 -30960.502} C_VEL
LIN {X 0,Y 257.057,Z 966.234,A -85,B 0,C 180,E1 -30961.475,E2 -30961.475} C_VEL
LIN {X 0,Y 238.269,Z 982.731,A -85,B 0,C 180,E1 -30962.854,E2 -30962.854} C_VEL
LIN {X 0,Y 219.646,Z 996.988,A -85,B 0,C 180,E1 -30964.478,E2 -30964.478} C_VEL
LIN {X 0,Y 199.577,Z 1010.714,A -85,B 0,C 180,E1 -30966.617,E2 -30966.617} C_VEL
LIN {X 0,Y 179.344,Z 1022.688,A -85,B 0,C 180,E1 -30969.311,E2 -30969.311} C_VEL
LIN {X 0,Y 160.881,Z 1032.406,A -85,B 0,C 180,E1 -30972.444,E2 -30972.444} C_VEL
LIN {X 0,Y 154.221,Z 1035.535,A -85,B 0,C 180,E1 -30973.36,E2 -30973.36} C_VEL
LIN {X 0,Y 135.787,Z 1042.77,A -85,B 0,C 180,E1 -30974.808,E2 -30974.808} C_VEL
LIN {X 0,Y 129.076,Z 1045.346,A -85,B 0,C 180,E1 -30976.065,E2 -30976.065} C_VEL
LIN {X 0,Y 108.601,Z 1052.605,A -85,B 0,C 180,E1 -30982.971,E2 -30982.971} C_VEL
LIN {X 0,Y 91.731,Z 1057.785,A -85,B 0,C 180,E1 -30991.764,E2 -30991.764} C_VEL
LIN {X 0,Y 75.353,Z 1062.165,A -85,B 0,C 180,E1 -31006.871,E2 -31006.871} C_VEL
LIN {X 0,Y 67.182,Z 1064.204,A -85,B 0,C 180,E1 -31022.524,E2 -31022.524} C_VEL
LIN {X 0,Y 64.136,Z 1065.073,A -85,B 0,C 180,E1 -31039.217,E2 -31039.217} C_VEL
LIN {X 0,Y 64.078,Z 1065.072,A -85,B 0,C 180,E1 -31050,E2 -31050} C_VEL
LIN {X 0,Y 64.18,Z 1064.608,A -85,B 0,C 180,E1 -31061.685,E2 -31061.685} C_VEL
LIN {X 0,Y 67.723,Z 1062.853,A -85,B 0,C 180,E1 -31079.158,E2 -31079.158} C_VEL
LIN {X 0,Y 76.546,Z 1059.824,A -85,B 0,C 180,E1 -31094.86,E2 -31094.86} C_VEL
LIN {X 0,Y 93.029,Z 1054.3,A -85,B 0,C 180,E1 -31109.3,E2 -31109.3} C_VEL
LIN {X 0,Y 109.254,Z 1048.329,A -85,B 0,C 180,E1 -31117.571,E2 -31117.571} C_VEL
LIN {X 0,Y 129.746,Z 1039.869,A -85,B 0,C 180,E1 -31124.432,E2 -31124.432} C_VEL
LIN {X 0,Y 148.777,Z 1030.765,A -85,B 0,C 180,E1 -31128.88,E2 -31128.88} C_VEL
LIN {X 0,Y 169.446,Z 1019.647,A -85,B 0,C 180,E1 -31132.46,E2 -31132.46} C_VEL
LIN {X 0,Y 189.75,Z 1006.955,A -85,B 0,C 180,E1 -31135.164,E2 -31135.164} C_VEL
LIN {X 0,Y 208.238,Z 994.002,A -85,B 0,C 180,E1 -31137.128,E2 -31137.128} C_VEL
LIN {X 0,Y 228.02,Z 978.178,A -85,B 0,C 180,E1 -31138.853,E2 -31138.853} C_VEL
LIN {X 0,Y 243.973,Z 963.826,A -85,B 0,C 180,E1 -31140.019,E2 -31140.019} C_VEL
LIN {X 0,Y 262.527,Z 944.959,A -85,B 0,C 180,E1 -31141.185,E2 -31141.185} C_VEL
LIN {X 0,Y 268.064,Z 938.779,A -85,B 0,C 180,E1 -31141.515,E2 -31141.515} C_VEL
LIN {X 0,Y 252.856,Z 954.951,A -85,B 0,C 180,E1 -31142.493,E2 -31142.493} C_VEL
LIN {X 0,Y 234.503,Z 972.265,A -85,B 0,C 180,E1 -31143.85,E2 -31143.85} C_VEL
LIN {X 0,Y 216.926,Z 986.762,A -85,B 0,C 180,E1 -31145.364,E2 -31145.364} C_VEL
LIN {X 0,Y 197.604,Z 1000.999,A -85,B 0,C 180,E1 -31147.355,E2 -31147.355} C_VEL
LIN {X 0,Y 177.615,Z 1013.715,A -85,B 0,C 180,E1 -31149.881,E2 -31149.881} C_VEL
LIN {X 0,Y 158.047,Z 1024.777,A -85,B 0,C 180,E1 -31153.022,E2 -31153.022} C_VEL
LIN {X 0,Y 137.276,Z 1034.875,A -85,B 0,C 180,E1 -31157.412,E2 -31157.412} C_VEL
LIN {X 0,Y 118.356,Z 1042.943,A -85,B 0,C 180,E1 -31162.95,E2 -31162.95} C_VEL
LIN {X 0,Y 98.584,Z 1050.194,A -85,B 0,C 180,E1 -31171.573,E2 -31171.573} C_VEL
LIN {X 0,Y 83.59,Z 1055.079,A -85,B 0,C 180,E1 -31182.13,E2 -31182.13} C_VEL
LIN {X 0,Y 70.513,Z 1059.076,A -85,B 0,C 180,E1 -31199.304,E2 -31199.304} C_VEL
LIN {X 0,Y 65.366,Z 1060.824,A -85,B 0,C 180,E1 -31214.928,E2 -31214.928} C_VEL
LIN {X 0,Y 64.106,Z 1061.577,A -85,B 0,C 180,E1 -31229.106,E2 -31229.106} C_VEL
LIN {X 0,Y 64.418,Z 1061.735,A -85,B 0,C 180,E1 -31241.642,E2 -31241.642} C_VEL
LIN {X 0,Y 67.808,Z 1061.092,A -85,B 0,C 180,E1 -31258.156,E2 -31258.156} C_VEL
LIN {X 0,Y 75.884,Z 1059.388,A -85,B 0,C 180,E1 -31273.25,E2 -31273.25} C_VEL
LIN {X 0,Y 90.701,Z 1055.888,A -85,B 0,C 180,E1 -31287.304,E2 -31287.304} C_VEL
LIN {X 0,Y 107.795,Z 1050.971,A -85,B 0,C 180,E1 -31296.681,E2 -31296.681} C_VEL
LIN {X 0,Y 128.058,Z 1044.244,A -85,B 0,C 180,E1 -31303.821,E2 -31303.821} C_VEL
LIN {X 0,Y 148.792,Z 1035.891,A -85,B 0,C 180,E1 -31308.852,E2 -31308.852} C_VEL
LIN {X 0,Y 169.6,Z 1026.27,A -85,B 0,C 180,E1 -31312.547,E2 -31312.547} C_VEL
LIN {X 0,Y 190.59,Z 1014.857,A -85,B 0,C 180,E1 -31315.413,E2 -31315.413} C_VEL
LIN {X 0,Y 210.259,Z 1002.709,A -85,B 0,C 180,E1 -31317.547,E2 -31317.547} C_VEL
LIN {X 0,Y 230.988,Z 987.939,A -85,B 0,C 180,E1 -31319.392,E2 -31319.392} C_VEL
LIN {X 0,Y 244.535,Z 977.131,A -85,B 0,C 180,E1 -31320.425,E2 -31320.425} C_VEL
LIN {X 0,Y 225.092,Z 992.64,A -85,B 0,C 180,E1 -31321.848,E2 -31321.848} C_VEL
LIN {X 0,Y 205.379,Z 1006.28,A -85,B 0,C 180,E1 -31323.585,E2 -31323.585} C_VEL
LIN {X 0,Y 184.167,Z 1019.311,A -85,B 0,C 180,E1 -31325.921,E2 -31325.921} C_VEL
LIN {X 0,Y 162.956,Z 1030.449,A -85,B 0,C 180,E1 -31328.926,E2 -31328.926} C_VEL
LIN {X 0,Y 141.601,Z 1040.317,A -85,B 0,C 180,E1 -31332.977,E2 -31332.977} C_VEL
LIN {X 0,Y 129.076,Z 1045.346,A -85,B 0,C 180,E1 -31336.065,E2 -31336.065} C_VEL
LIN {X 0,Y 122.389,Z 1047.811,A -85,B 0,C 180,E1 -31337.471,E2 -31337.471} C_VEL
LIN {X 0,Y 102.768,Z 1053.524,A -85,B 0,C 180,E1 -31340.457,E2 -31340.457} C_VEL
LIN {X 0,Y 97.131,Z 1055.053,A -85,B 0,C 180,E1 -31342.3,E2 -31342.3} C_VEL
LIN {X 0,Y 78.848,Z 1059.803,A -85,B 0,C 180,E1 -31353.179,E2 -31353.179} C_VEL
LIN {X 0,Y 65.517,Z 1062.863,A -85,B 0,C 180,E1 -31367.816,E2 -31367.816} C_VEL
LIN {X 0,Y 57.203,Z 1064.641,A -85,B 0,C 180,E1 -31389.538,E2 -31389.538} C_VEL
LIN {X 0,Y 56.02,Z 1064.939,A -85,B 0,C 180,E1 -31405.906,E2 -31405.906} C_VEL
LIN {X 0,Y 56.018,Z 1064.736,A -85,B 0,C 180,E1 -31415.12,E2 -31415.12} C_VEL
LIN {X 0,Y 57.802,Z 1063.651,A -85,B 0,C 180,E1 -31433.535,E2 -31433.535} C_VEL
LIN {X 0,Y 67.524,Z 1060.58,A -85,B 0,C 180,E1 -31455.299,E2 -31455.299} C_VEL
LIN {X 0,Y 81.292,Z 1056.486,A -85,B 0,C 180,E1 -31468.896,E2 -31468.896} C_VEL
LIN {X 0,Y 101.484,Z 1049.849,A -85,B 0,C 180,E1 -31479.828,E2 -31479.828} C_VEL
LIN {X 0,Y 120.485,Z 1042.59,A -85,B 0,C 180,E1 -31486.159,E2 -31486.159} C_VEL
LIN {X 0,Y 142.668,Z 1032.818,A -85,B 0,C 180,E1 -31491.188,E2 -31491.188} C_VEL
LIN {X 0,Y 162.74,Z 1022.5,A -85,B 0,C 180,E1 -31494.467,E2 -31494.467} C_VEL
LIN {X 0,Y 184.211,Z 1009.932,A -85,B 0,C 180,E1 -31497.129,E2 -31497.129} C_VEL
LIN {X 0,Y 204.005,Z 996.526,A -85,B 0,C 180,E1 -31499.062,E2 -31499.062} C_VEL
LIN {X 0,Y 223.989,Z 981.263,A -85,B 0,C 180,E1 -31500.639,E2 -31500.639} C_VEL
LIN {X 0,Y 238.066,Z 969.095,A -85,B 0,C 180,E1 -31501.601,E2 -31501.601} C_VEL
LIN {X 0,Y 218.288,Z 985.57,A -85,B 0,C 180,E1 -31503.065,E2 -31503.065} C_VEL
LIN {X 0,Y 200.631,Z 998.563,A -85,B 0,C 180,E1 -31504.624,E2 -31504.624} C_VEL
LIN {X 0,Y 178.323,Z 1012.889,A -85,B 0,C 180,E1 -31507.036,E2 -31507.036} C_VEL
LIN {X 0,Y 159.241,Z 1023.553,A -85,B 0,C 180,E1 -31509.662,E2 -31509.662} C_VEL
LIN {X 0,Y 136.887,Z 1034.358,A -85,B 0,C 180,E1 -31513.714,E2 -31513.714} C_VEL
LIN {X 0,Y 118.037,Z 1042.176,A -85,B 0,C 180,E1 -31518.424,E2 -31518.424} C_VEL
LIN {X 0,Y 96.962,Z 1049.707,A -85,B 0,C 180,E1 -31526.213,E2 -31526.213} C_VEL
LIN {X 0,Y 80.417,Z 1054.726,A -85,B 0,C 180,E1 -31536.08,E2 -31536.08} C_VEL
LIN {X 0,Y 66.011,Z 1058.76,A -85,B 0,C 180,E1 -31551.608,E2 -31551.608} C_VEL
LIN {X 0,Y 57.807,Z 1060.995,A -85,B 0,C 180,E1 -31572.053,E2 -31572.053} C_VEL
LIN {X 0,Y 56.124,Z 1061.772,A -85,B 0,C 180,E1 -31587.958,E2 -31587.958} C_VEL
LIN {X 0,Y 56.368,Z 1061.987,A -85,B 0,C 180,E1 -31601.252,E2 -31601.252} C_VEL
LIN {X 0,Y 60.39,Z 1061.363,A -85,B 0,C 180,E1 -31620.882,E2 -31620.882} C_VEL
LIN {X 0,Y 70.121,Z 1059.591,A -85,B 0,C 180,E1 -31637.859,E2 -31637.859} C_VEL
LIN {X 0,Y 87.01,Z 1055.945,A -85,B 0,C 180,E1 -31652.234,E2 -31652.234} C_VEL
LIN {X 0,Y 105.641,Z 1050.907,A -85,B 0,C 180,E1 -31661.174,E2 -31661.174} C_VEL
LIN {X 0,Y 126.912,Z 1044.079,A -85,B 0,C 180,E1 -31667.674,E2 -31667.674} C_VEL
LIN {X 0,Y 148.361,Z 1035.653,A -85,B 0,C 180,E1 -31672.186,E2 -31672.186} C_VEL
LIN {X 0,Y 169.517,Z 1026.05,A -85,B 0,C 180,E1 -31675.443,E2 -31675.443} C_VEL
LIN {X 0,Y 191.095,Z 1014.425,A -85,B 0,C 180,E1 -31678,E2 -31678} C_VEL
LIN {X 0,Y 211.977,Z 1001.629,A -85,B 0,C 180,E1 -31679.954,E2 -31679.954} C_VEL
LIN {X 0,Y 216.699,Z 998.359,A -85,B 0,C 180,E1 -31680.349,E2 -31680.349} C_VEL
LIN {X 0,Y 194.132,Z 1012.942,A -85,B 0,C 180,E1 -31682.274,E2 -31682.274} C_VEL
LIN {X 0,Y 174.491,Z 1023.956,A -85,B 0,C 180,E1 -31684.384,E2 -31684.384} C_VEL
LIN {X 0,Y 151.327,Z 1035.224,A -85,B 0,C 180,E1 -31687.641,E2 -31687.641} C_VEL
LIN {X 0,Y 131.587,Z 1043.397,A -85,B 0,C 180,E1 -31691.411,E2 -31691.411} C_VEL
LIN {X 0,Y 109.971,Z 1051.117,A -85,B 0,C 180,E1 -31697.313,E2 -31697.313} C_VEL
LIN {X 0,Y 97.131,Z 1055.053,A -85,B 0,C 180,E1 -31702.3,E2 -31702.3} C_VEL
LIN {X 0,Y 90.61,Z 1056.71,A -85,B 0,C 180,E1 -31704.674,E2 -31704.674} C_VEL
LIN {X 0,Y 71.631,Z 1060.476,A -85,B 0,C 180,E1 -31710.945,E2 -31710.945} C_VEL
LIN {X 0,Y 66.583,Z 1061.353,A -85,B 0,C 180,E1 -31714.487,E2 -31714.487} C_VEL
LIN {X 0,Y 53.633,Z 1063.713,A -85,B 0,C 180,E1 -31733.374,E2 -31733.374} C_VEL
LIN {X 0,Y 48.448,Z 1064.62,A -85,B 0,C 180,E1 -31754.437,E2 -31754.437} C_VEL
LIN {X 0,Y 48.06,Z 1064.66,A -85,B 0,C 180,E1 -31768.808,E2 -31768.808} C_VEL
LIN {X 0,Y 48.232,Z 1064.311,A -85,B 0,C 180,E1 -31783.006,E2 -31783.006} C_VEL
LIN {X 0,Y 53.586,Z 1062.502,A -85,B 0,C 180,E1 -31806.663,E2 -31806.663} C_VEL
LIN {X 0,Y 65.293,Z 1059.487,A -85,B 0,C 180,E1 -31824.414,E2 -31824.414} C_VEL
LIN {X 0,Y 84.1,Z 1054.308,A -85,B 0,C 180,E1 -31838.027,E2 -31838.027} C_VEL
LIN {X 0,Y 103.157,Z 1048.11,A -85,B 0,C 180,E1 -31845.764,E2 -31845.764} C_VEL
LIN {X 0,Y 125.358,Z 1039.722,A -85,B 0,C 180,E1 -31851.516,E2 -31851.516} C_VEL
LIN {X 0,Y 146.483,Z 1030.188,A -85,B 0,C 180,E1 -31855.266,E2 -31855.266} C_VEL
LIN {X 0,Y 168.076,Z 1019.049,A -85,B 0,C 180,E1 -31858.076,E2 -31858.076} C_VEL
LIN {X 0,Y 188.98,Z 1006.39,A -85,B 0,C 180,E1 -31860.162,E2 -31860.162} C_VEL
LIN {X 0,Y 207.823,Z 993.527,A -85,B 0,C 180,E1 -31861.689,E2 -31861.689} C_VEL
LIN {X 0,Y 189.285,Z 1006.002,A -85,B 0,C 180,E1 -31863.258,E2 -31863.258} C_VEL
LIN {X 0,Y 168.439,Z 1018.428,A -85,B 0,C 180,E1 -31865.45,E2 -31865.45} C_VEL
LIN {X 0,Y 147.516,Z 1029.03,A -85,B 0,C 180,E1 -31868.265,E2 -31868.265} C_VEL
LIN {X 0,Y 126.765,Z 1038.203,A -85,B 0,C 180,E1 -31872.02,E2 -31872.02} C_VEL
LIN {X 0,Y 104.937,Z 1046.277,A -85,B 0,C 180,E1 -31877.665,E2 -31877.665} C_VEL
LIN {X 0,Y 86.145,Z 1052.186,A -85,B 0,C 180,E1 -31885.129,E2 -31885.129} C_VEL
LIN {X 0,Y 66.651,Z 1057.312,A -85,B 0,C 180,E1 -31898.731,E2 -31898.731} C_VEL
LIN {X 0,Y 54.829,Z 1060.084,A -85,B 0,C 180,E1 -31915.575,E2 -31915.575} C_VEL
LIN {X 0,Y 48.729,Z 1061.727,A -85,B 0,C 180,E1 -31938.159,E2 -31938.159} C_VEL
LIN {X 0,Y 48.068,Z 1062.103,A -85,B 0,C 180,E1 -31953.578,E2 -31953.578} C_VEL
LIN {X 0,Y 49.156,Z 1062.102,A -85,B 0,C 180,E1 -31968.993,E2 -31968.993} C_VEL
LIN {X 0,Y 55.293,Z 1061.319,A -85,B 0,C 180,E1 -31989.266,E2 -31989.266} C_VEL
LIN {X 0,Y 69.814,Z 1058.978,A -85,B 0,C 180,E1 -32008,E2 -32008} C_VEL
LIN {X 0,Y 88.457,Z 1054.931,A -85,B 0,C 180,E1 -32019.752,E2 -32019.752} C_VEL
LIN {X 0,Y 109.601,Z 1049.347,A -85,B 0,C 180,E1 -32027.464,E2 -32027.464} C_VEL
LIN {X 0,Y 131.092,Z 1042.163,A -85,B 0,C 180,E1 -32032.551,E2 -32032.551} C_VEL
LIN {X 0,Y 152.337,Z 1033.816,A -85,B 0,C 180,E1 -32036.096,E2 -32036.096} C_VEL
LIN {X 0,Y 175.013,Z 1023.147,A -85,B 0,C 180,E1 -32038.908,E2 -32038.908} C_VEL
LIN {X 0,Y 188.564,Z 1015.938,A -85,B 0,C 180,E1 -32040.297,E2 -32040.297} C_VEL
LIN {X 0,Y 165.157,Z 1028.282,A -85,B 0,C 180,E1 -32042.64,E2 -32042.64} C_VEL
LIN {X 0,Y 144.618,Z 1037.527,A -85,B 0,C 180,E1 -32045.368,E2 -32045.368} C_VEL
LIN {X 0,Y 121.687,Z 1046.35,A -85,B 0,C 180,E1 -32049.59,E2 -32049.59} C_VEL
LIN {X 0,Y 100.58,Z 1053.019,A -85,B 0,C 180,E1 -32055.355,E2 -32055.355} C_VEL
LIN {X 0,Y 79.333,Z 1058.608,A -85,B 0,C 180,E1 -32064.842,E2 -32064.842} C_VEL
LIN {X 0,Y 66.583,Z 1061.353,A -85,B 0,C 180,E1 -32074.487,E2 -32074.487} C_VEL
LIN {X 0,Y 60.946,Z 1062.254,A -85,B 0,C 180,E1 -32079.227,E2 -32079.227} C_VEL
LIN {X 0,Y 48.828,Z 1063.644,A -85,B 0,C 180,E1 -32089.603,E2 -32089.603} C_VEL
LIN {X 0,Y 43.169,Z 1064.164,A -85,B 0,C 180,E1 -32099.121,E2 -32099.121} C_VEL
LIN {X 0,Y 42.163,Z 1064.23,A -85,B 0,C 180,E1 -32102.614,E2 -32102.614} C_VEL
LIN {X 0,Y 40.022,Z 1064.484,A -85,B 0,C 180,E1 -32125.701,E2 -32125.701} C_VEL
LIN {X 0,Y 40.03,Z 1064.301,A -85,B 0,C 180,E1 -32137.174,E2 -32137.174} C_VEL
LIN {X 0,Y 44.07,Z 1063.056,A -85,B 0,C 180,E1 -32164.556,E2 -32164.556} C_VEL
LIN {X 0,Y 57.857,Z 1059.928,A -85,B 0,C 180,E1 -32187.867,E2 -32187.867} C_VEL
LIN {X 0,Y 74.437,Z 1055.902,A -85,B 0,C 180,E1 -32200.099,E2 -32200.099} C_VEL
LIN {X 0,Y 97.698,Z 1049.091,A -85,B 0,C 180,E1 -32209.269,E2 -32209.269} C_VEL
LIN {X 0,Y 117.622,Z 1042.044,A -85,B 0,C 180,E1 -32214.043,E2 -32214.043} C_VEL
LIN {X 0,Y 141.082,Z 1032.241,A -85,B 0,C 180,E1 -32217.869,E2 -32217.869} C_VEL
LIN {X 0,Y 160.983,Z 1022.432,A -85,B 0,C 180,E1 -32220.215,E2 -32220.215} C_VEL
LIN {X 0,Y 177.521,Z 1013.232,A -85,B 0,C 180,E1 -32221.752,E2 -32221.752} C_VEL
LIN {X 0,Y 158.31,Z 1023.632,A -85,B 0,C 180,E1 -32223.687,E2 -32223.687} C_VEL
LIN {X 0,Y 134.501,Z 1034.689,A -85,B 0,C 180,E1 -32226.831,E2 -32226.831} C_VEL
LIN {X 0,Y 114.879,Z 1042.369,A -85,B 0,C 180,E1 -32230.411,E2 -32230.411} C_VEL
LIN {X 0,Y 92.738,Z 1049.722,A -85,B 0,C 180,E1 -32236.346,E2 -32236.346} C_VEL
LIN {X 0,Y 72.424,Z 1055.127,A -85,B 0,C 180,E1 -32245.34,E2 -32245.34} C_VEL
LIN {X 0,Y 54.254,Z 1059.23,A -85,B 0,C 180,E1 -32260.92,E2 -32260.92} C_VEL
LIN {X 0,Y 42.848,Z 1061.432,A -85,B 0,C 180,E1 -32285.163,E2 -32285.163} C_VEL
LIN {X 0,Y 40.142,Z 1062.206,A -85,B 0,C 180,E1 -32307.145,E2 -32307.145} C_VEL
LIN {X 0,Y 40.672,Z 1062.41,A -85,B 0,C 180,E1 -32325.69,E2 -32325.69} C_VEL
LIN {X 0,Y 47.124,Z 1061.779,A -85,B 0,C 180,E1 -32351.13,E2 -32351.13} C_VEL
LIN {X 0,Y 60.323,Z 1059.997,A -85,B 0,C 180,E1 -32369.535,E2 -32369.535} C_VEL
LIN {X 0,Y 80.642,Z 1056.326,A -85,B 0,C 180,E1 -32382.695,E2 -32382.695} C_VEL
LIN {X 0,Y 100.575,Z 1051.523,A -85,B 0,C 180,E1 -32389.81,E2 -32389.81} C_VEL
LIN {X 0,Y 123.46,Z 1044.763,A -85,B 0,C 180,E1 -32394.982,E2 -32394.982} C_VEL
LIN {X 0,Y 146.036,Z 1036.376,A -85,B 0,C 180,E1 -32398.475,E2 -32398.475} C_VEL
LIN {X 0,Y 160.608,Z 1030.16,A -85,B 0,C 180,E1 -32400.196,E2 -32400.196} C_VEL
LIN {X 0,Y 137.175,Z 1040.182,A -85,B 0,C 180,E1 -32403.019,E2 -32403.019} C_VEL
LIN {X 0,Y 114.802,Z 1048.029,A -85,B 0,C 180,E1 -32406.828,E2 -32406.828} C_VEL
LIN {X 0,Y 92.243,Z 1054.65,A -85,B 0,C 180,E1 -32412.689,E2 -32412.689} C_VEL
LIN {X 0,Y 71.164,Z 1059.409,A -85,B 0,C 180,E1 -32421.976,E2 -32421.976} C_VEL
LIN {X 0,Y 53.808,Z 1062.577,A -85,B 0,C 180,E1 -32436.96,E2 -32436.96} C_VEL
LIN {X 0,Y 42.163,Z 1064.23,A -85,B 0,C 180,E1 -32462.614,E2 -32462.614} C_VEL
LIN {X 0,Y 39.826,Z 1064.407,A -85,B 0,C 180,E1 -32471.332,E2 -32471.332} C_VEL
LIN {X 0,Y 36.217,Z 1064.401,A -85,B 0,C 180,E1 -32483.726,E2 -32483.726} C_VEL
LIN {X 0,Y 33.295,Z 1063.674,A -85,B 0,C 180,E1 -32513.967,E2 -32513.967} C_VEL
LIN {X 0,Y 33.85,Z 1063.503,A -85,B 0,C 180,E1 -32517.766,E2 -32517.766} C_VEL
LIN {X 0,Y 43.543,Z 1061.673,A -85,B 0,C 180,E1 -32543.487,E2 -32543.487} C_VEL
LIN {X 0,Y 62.284,Z 1058.004,A -85,B 0,C 180,E1 -32561.292,E2 -32561.292} C_VEL
LIN {X 0,Y 84.085,Z 1052.48,A -85,B 0,C 180,E1 -32570.747,E2 -32570.747} C_VEL
LIN {X 0,Y 107.202,Z 1045.387,A -85,B 0,C 180,E1 -32576.378,E2 -32576.378} C_VEL
LIN {X 0,Y 130.471,Z 1036.475,A -85,B 0,C 180,E1 -32580,E2 -32580} C_VEL
LIN {X 0,Y 146.709,Z 1029.307,A -85,B 0,C 180,E1 -32581.839,E2 -32581.839} C_VEL
LIN {X 0,Y 125.373,Z 1038.359,A -85,B 0,C 180,E1 -32584.502,E2 -32584.502} C_VEL
LIN {X 0,Y 102.142,Z 1046.505,A -85,B 0,C 180,E1 -32588.617,E2 -32588.617} C_VEL
LIN {X 0,Y 81.502,Z 1052.448,A -85,B 0,C 180,E1 -32594.258,E2 -32594.258} C_VEL
LIN {X 0,Y 58.712,Z 1057.638,A -85,B 0,C 180,E1 -32605.497,E2 -32605.497} C_VEL
LIN {X 0,Y 42.738,Z 1060.505,A -85,B 0,C 180,E1 -32622.726,E2 -32622.726} C_VEL
LIN {X 0,Y 33.191,Z 1062.175,A -85,B 0,C 180,E1 -32652.467,E2 -32652.467} C_VEL
LIN {X 0,Y 32.075,Z 1062.519,A -85,B 0,C 180,E1 -32674.005,E2 -32674.005} C_VEL
LIN {X 0,Y 33.931,Z 1062.547,A -85,B 0,C 180,E1 -32696.233,E2 -32696.233} C_VEL
LIN {X 0,Y 43.2,Z 1061.799,A -85,B 0,C 180,E1 -32721.902,E2 -32721.902} C_VEL
LIN {X 0,Y 61.616,Z 1059.549,A -85,B 0,C 180,E1 -32740.256,E2 -32740.256} C_VEL
LIN {X 0,Y 83.233,Z 1055.513,A -85,B 0,C 180,E1 -32750.09,E2 -32750.09} C_VEL
LIN {X 0,Y 105.277,Z 1050.216,A -85,B 0,C 180,E1 -32755.761,E2 -32755.761} C_VEL
LIN {X 0,Y 128.988,Z 1042.849,A -85,B 0,C 180,E1 -32759.687,E2 -32759.687} C_VEL
LIN {X 0,Y 132.228,Z 1041.722,A -85,B 0,C 180,E1 -32760.114,E2 -32760.114} C_VEL
LIN {X 0,Y 111.161,Z 1048.78,A -85,B 0,C 180,E1 -32763.194,E2 -32763.194} C_VEL
LIN {X 0,Y 86.03,Z 1055.529,A -85,B 0,C 180,E1 -32768.914,E2 -32768.914} C_VEL
LIN {X 0,Y 65.839,Z 1059.71,A -85,B 0,C 180,E1 -32776.907,E2 -32776.907} C_VEL
LIN {X 0,Y 44.951,Z 1062.924,A -85,B 0,C 180,E1 -32794.611,E2 -32794.611} C_VEL
LIN {X 0,Y 33.94,Z 1064.111,A -85,B 0,C 180,E1 -32821.877,E2 -32821.877} C_VEL
LIN {X 0,Y 32.036,Z 1064.238,A -85,B 0,C 180,E1 -32847.139,E2 -32847.139} C_VEL
LIN {X 0,Y 32.254,Z 1064.005,A -85,B 0,C 180,E1 -32864.359,E2 -32864.359} C_VEL
LIN {X 0,Y 33.85,Z 1063.503,A -85,B 0,C 180,E1 -32877.766,E2 -32877.766} C_VEL
LIN {X 0,Y 35.925,Z 1062.949,A -85,B 0,C 180,E1 -32890.032,E2 -32890.032} C_VEL
LIN {X 0,Y 45.545,Z 1060.543,A -85,B 0,C 180,E1 -32918.823,E2 -32918.823} C_VEL
LIN {X 0,Y 49.862,Z 1059.662,A -85,B 0,C 180,E1 -32922.955,E2 -32922.955} C_VEL
LIN {X 0,Y 69.78,Z 1055.57,A -85,B 0,C 180,E1 -32932.59,E2 -32932.59} C_VEL
LIN {X 0,Y 95.008,Z 1048.871,A -85,B 0,C 180,E1 -32938.87,E2 -32938.87} C_VEL
LIN {X 0,Y 115.31,Z 1042.129,A -85,B 0,C 180,E1 -32941.944,E2 -32941.944} C_VEL
LIN {X 0,Y 92.442,Z 1049.426,A -85,B 0,C 180,E1 -32945.671,E2 -32945.671} C_VEL
LIN {X 0,Y 69.46,Z 1055.115,A -85,B 0,C 180,E1 -32951.798,E2 -32951.798} C_VEL
LIN {X 0,Y 49.554,Z 1058.954,A -85,B 0,C 180,E1 -32961.847,E2 -32961.847} C_VEL
LIN {X 0,Y 30.708,Z 1061.689,A -85,B 0,C 180,E1 -32986.86,E2 -32986.86} C_VEL
LIN {X 0,Y 24.252,Z 1062.618,A -85,B 0,C 180,E1 -33022.896,E2 -33022.896} C_VEL
LIN {X 0,Y 24.751,Z 1062.878,A -85,B 0,C 180,E1 -33048.856,E2 -33048.856} C_VEL
LIN {X 0,Y 35.699,Z 1062.259,A -85,B 0,C 180,E1 -33087.17,E2 -33087.17} C_VEL
LIN {X 0,Y 52.977,Z 1060.511,A -85,B 0,C 180,E1 -33104.278,E2 -33104.278} C_VEL
LIN {X 0,Y 75.417,Z 1057.108,A -85,B 0,C 180,E1 -33113.914,E2 -33113.914} C_VEL
LIN {X 0,Y 98.997,Z 1051.89,A -85,B 0,C 180,E1 -33119.296,E2 -33119.296} C_VEL
LIN {X 0,Y 103.102,Z 1050.871,A -85,B 0,C 180,E1 -33120.049,E2 -33120.049} C_VEL
LIN {X 0,Y 81.222,Z 1056.191,A -85,B 0,C 180,E1 -33124.321,E2 -33124.321} C_VEL
LIN {X 0,Y 57.411,Z 1060.608,A -85,B 0,C 180,E1 -33132.754,E2 -33132.754} C_VEL
LIN {X 0,Y 37.703,Z 1063.012,A -85,B 0,C 180,E1 -33148.934,E2 -33148.934} C_VEL
LIN {X 0,Y 25.85,Z 1063.981,A -85,B 0,C 180,E1 -33179.811,E2 -33179.811} C_VEL
LIN {X 0,Y 24.073,Z 1063.988,A -85,B 0,C 180,E1 -33210,E2 -33210} C_VEL
LIN {X 0,Y 26.511,Z 1063.347,A -85,B 0,C 180,E1 -33243.926,E2 -33243.926} C_VEL
LIN {X 0,Y 39.216,Z 1061.438,A -85,B 0,C 180,E1 -33273.175,E2 -33273.175} C_VEL
LIN {X 0,Y 49.862,Z 1059.662,A -85,B 0,C 180,E1 -33282.955,E2 -33282.955} C_VEL
LIN {X 0,Y 56.049,Z 1058.451,A -85,B 0,C 180,E1 -33287.862,E2 -33287.862} C_VEL
LIN {X 0,Y 72.98,Z 1054.561,A -85,B 0,C 180,E1 -33299.722,E2 -33299.722} C_VEL
LIN {X 0,Y 78.536,Z 1053.138,A -85,B 0,C 180,E1 -33301.336,E2 -33301.336} C_VEL
LIN {X 0,Y 82.675,Z 1052.06,A -85,B 0,C 180,E1 -33302.079,E2 -33302.079} C_VEL
LIN {X 0,Y 58.551,Z 1057.348,A -85,B 0,C 180,E1 -33307.916,E2 -33307.916} C_VEL
LIN {X 0,Y 36.185,Z 1060.687,A -85,B 0,C 180,E1 -33320.033,E2 -33320.033} C_VEL
LIN {X 0,Y 21.273,Z 1062.299,A -85,B 0,C 180,E1 -33345.169,E2 -33345.169} C_VEL
LIN {X 0,Y 16.14,Z 1062.878,A -85,B 0,C 180,E1 -33386.449,E2 -33386.449} C_VEL
LIN {X 0,Y 18.509,Z 1063.048,A -85,B 0,C 180,E1 -33426.459,E2 -33426.459} C_VEL
LIN {X 0,Y 32.871,Z 1062.405,A -85,B 0,C 180,E1 -33460.556,E2 -33460.556} C_VEL
LIN {X 0,Y 52.324,Z 1060.607,A -85,B 0,C 180,E1 -33473.57,E2 -33473.57} C_VEL
LIN {X 0,Y 73.451,Z 1057.574,A -85,B 0,C 180,E1 -33479.888,E2 -33479.888} C_VEL
LIN {X 0,Y 50.122,Z 1061.154,A -85,B 0,C 180,E1 -33486.874,E2 -33486.874} C_VEL
LIN {X 0,Y 30.141,Z 1063.174,A -85,B 0,C 180,E1 -33501.74,E2 -33501.74} C_VEL
LIN {X 0,Y 16.511,Z 1063.886,A -85,B 0,C 180,E1 -33548.694,E2 -33548.694} C_VEL
LIN {X 0,Y 16.029,Z 1063.747,A -85,B 0,C 180,E1 -33573.576,E2 -33573.576} C_VEL
LIN {X 0,Y 21.014,Z 1063.032,A -85,B 0,C 180,E1 -33619.579,E2 -33619.579} C_VEL
LIN {X 0,Y 37.164,Z 1061.082,A -85,B 0,C 180,E1 -33645.597,E2 -33645.597} C_VEL
LIN {X 0,Y 61.062,Z 1057.076,A -85,B 0,C 180,E1 -33657.273,E2 -33657.273} C_VEL
LIN {X 0,Y 78.536,Z 1053.138,A -85,B 0,C 180,E1 -33661.336,E2 -33661.336} C_VEL
LIN {X 0,Y 76.859,Z 1053.554,A -85,B 0,C 180,E1 -33662.047,E2 -33662.047} C_VEL
LIN {X 0,Y 67.644,Z 1055.539,A -85,B 0,C 180,E1 -33662.616,E2 -33662.616} C_VEL
LIN {X 0,Y 48.871,Z 1059.025,A -85,B 0,C 180,E1 -33661.586,E2 -33661.586} C_VEL
LIN {X 0,Y 36.149,Z 1060.829,A -85,B 0,C 180,E1 -33658.441,E2 -33658.441} C_VEL
LIN {X 0,Y 16.908,Z 1062.805,A -85,B 0,C 180,E1 -33641.12,E2 -33641.12} C_VEL
LIN {X 0,Y 8.025,Z 1063.538,A -85,B 0,C 180,E1 -33574.641,E2 -33574.641} C_VEL
LIN {X 0,Y 13.539,Z 1063.581,A -85,B 0,C 180,E1 -33507.595,E2 -33507.595} C_VEL
LIN {X 0,Y 32.306,Z 1062.649,A -85,B 0,C 180,E1 -33483.549,E2 -33483.549} C_VEL
LIN {X 0,Y 41.628,Z 1061.928,A -85,B 0,C 180,E1 -33479.68,E2 -33479.68} C_VEL
LIN {X 0,Y 18.822,Z 1063.133,A -85,B 0,C 180,E1 -33462.983,E2 -33462.983} C_VEL
LIN {X 0,Y 8.44,Z 1063.189,A -85,B 0,C 180,E1 -33410.82,E2 -33410.82} C_VEL
LIN {X 0,Y 10.496,Z 1062.969,A -85,B 0,C 180,E1 -33348.177,E2 -33348.177} C_VEL
LIN {X 0,Y 29.443,Z 1061.463,A -85,B 0,C 180,E1 -33309.985,E2 -33309.985} C_VEL
LIN {X 0,Y 47.59,Z 1059.195,A -85,B 0,C 180,E1 -33302.237,E2 -33302.237} C_VEL
LIN {X 0,Y 36.149,Z 1060.829,A -85,B 0,C 180,E1 -33298.441,E2 -33298.441} C_VEL
LIN {X 0,Y 26.677,Z 1061.947,A -85,B 0,C 180,E1 -33295.181,E2 -33295.181} C_VEL
LIN {X 0,Y 13.532,Z 1062.899,A -85,B 0,C 180,E1 -33293.068,E2 -33293.068} C_VEL
LIN {X 0,Y 0.342,Z 1063.344,A -85,B 0,C 180,E1 -33119.688,E2 -33119.688} C_VEL
LIN {X 0,Y 0.649,Z 1063.35,A -85,B 0,C 180,E1 -33116.966,E2 -33116.966} C_VEL
LIN {X 0,Y 1.003,Z 1063.312,A -85,B 0,C 180,E1 -32944.426,E2 -32944.426} C_VEL
LIN {X 0,Y 0.342,Z 1063.344,A -85,B 0,C 180,E1 -33119.688,E2 -33119.688} C_VEL
LIN {X 0,Y 2.302,Z 1065.344,A -85,B 0,C 180,E1 -33114.794,E2 -33114.794} C_VEL
LIN {X 0,Y 2.302,Z 1088.5,A -85,B 0,C 180,E1 -33114.794,E2 -33114.794} C_VEL
LIN {X 0,Y 2.302,Z 1088.5,A -85,B 0,C 180,E1 -33114.794,E2 -33114.794}

QRS_NEXT_CUT()

QRS_NEXT()
QRS_HOME()

END
